Yaskawa INFORM job: test_long_tjr6.JBI

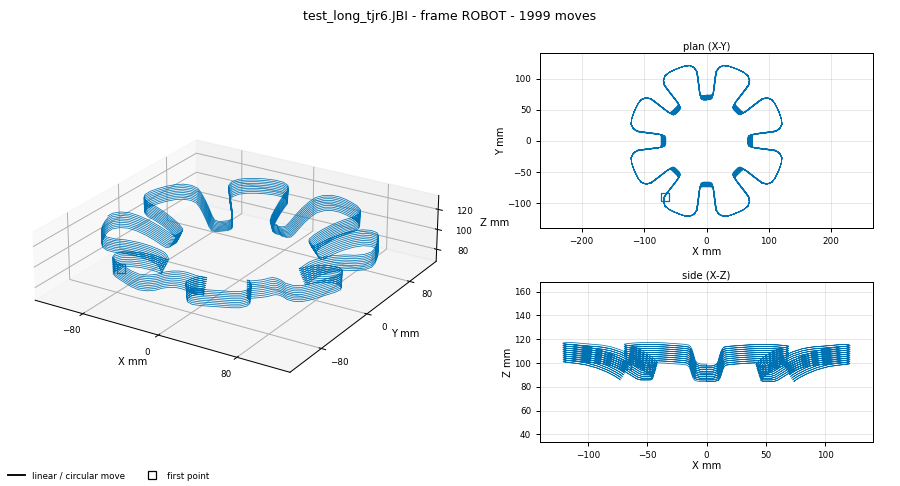
[picture p0: tool path of test_long_tjr6.JBI in frame ROBOT, 1999 of 2000 moves have a stored position in this frame; points joined in program order, loops and branches not executed]
version: 0
/JOB
//NAME test_long
//POS
///NPOS 48,0,0,2,0,0
///TOOL 1
///POSTYPE ROBOT
///RECTAN
///RCONF 1,0,0,0,0,0,0,0,0,0,0,0,0,0,0,0,0,0,0,0,0,0,0,0
C00000=-62.110,-83.210,96.990,-0.0900,0.0600,0.9900
C00001=-67.170,-90.300,98.220,-0.0900,0.0500,0.9900
C00002=-68.520,-97.840,98.870,-0.0700,-0.0100,1.0000
C00003=-65.820,-104.830,99.390,-0.0300,-0.0200,1.0000
C00004=-59.610,-109.840,99.910,-0.0000,-0.0000,1.0000
C00005=-51.890,-113.720,100.250,-0.0000,-0.0000,1.0000
C00006=-43.720,-117.100,100.250,-0.0000,-0.0000,1.0000
C00007=-35.520,-119.820,99.910,-0.0000,-0.0000,1.0000
C00008=-27.590,-120.670,99.390,0.0000,-0.0300,1.0000
C00009=-20.730,-117.630,98.870,0.0400,-0.0500,1.0000
C00010=-16.350,-111.350,98.220,0.1000,-0.0300,0.9900
C00011=-14.920,-102.760,96.990,0.1000,-0.0200,0.9900
C00012=-13.710,-93.380,94.450,0.0900,-0.0100,1.0000
C00013=-12.630,-84.870,91.070,0.0700,-0.0100,1.0000
C00014=-11.600,-78.400,87.740,0.0300,-0.0100,1.0000
C00015=-9.810,-74.590,85.320,-0.2400,0.2600,0.9300
C00016=-5.850,-73.580,84.360,-0.0500,0.5500,0.8400
C00017=-2.550,-73.670,84.320,0.0200,0.5600,0.8300
C00018=0.000,-73.710,84.350,-0.0000,0.5600,0.8300
C00019=0.000,-73.710,84.350,-0.0000,0.5600,0.8300
C00020=2.550,-73.670,84.320,-0.0200,0.5600,0.8300
C00021=5.850,-73.580,84.360,0.0500,0.5500,0.8400
C00022=9.810,-74.580,85.320,0.2400,0.2600,0.9300
C00023=11.600,-78.400,87.740,-0.0300,-0.0100,1.0000
C00024=12.630,-84.870,91.070,-0.0700,-0.0100,1.0000
C00025=13.710,-93.380,94.450,-0.0900,-0.0100,1.0000
C00026=14.920,-102.760,96.990,-0.1000,-0.0200,0.9900
C00027=16.350,-111.350,98.220,-0.1000,-0.0300,0.9900
C00028=20.730,-117.630,98.870,-0.0400,-0.0500,1.0000
C00029=27.590,-120.670,99.390,-0.0000,-0.0300,1.0000
C00030=35.520,-119.820,99.910,0.0000,-0.0000,1.0000
C00031=43.720,-117.100,100.250,0.0000,-0.0000,1.0000
C00032=51.890,-113.720,100.250,0.0000,-0.0000,1.0000
C00033=59.610,-109.840,99.910,0.0000,-0.0000,1.0000
C00034=65.820,-104.830,99.390,0.0300,-0.0200,1.0000
C00035=68.520,-97.840,98.870,0.0700,-0.0100,1.0000
C00036=67.170,-90.300,98.220,0.0900,0.0500,0.9900
C00037=62.110,-83.210,96.990,0.0900,0.0600,0.9900
C00038=56.330,-75.720,94.450,0.0800,0.0600,1.0000
C00039=51.080,-68.940,91.070,0.0600,0.0400,1.0000
C00040=47.240,-63.640,87.740,0.0200,0.0100,1.0000
C00041=45.800,-59.680,85.320,-0.3600,0.0200,0.9300
C00042=47.890,-56.170,84.360,-0.4200,0.3500,0.8400
C00043=50.290,-53.900,84.320,-0.3800,0.4100,0.8300
C00044=52.120,-52.120,84.350,-0.4000,0.4000,0.8300
C00045=53.900,-50.290,84.320,-0.4100,0.3800,0.8300
C00046=56.170,-47.890,84.360,-0.3500,0.4200,0.8400
C00047=59.680,-45.800,85.320,-0.0200,0.3600,0.9300
C00048=63.640,-47.240,87.740,-0.0100,-0.0200,1.0000
C00049=68.940,-51.080,91.070,-0.0400,-0.0600,1.0000
C00050=75.720,-56.330,94.450,-0.0600,-0.0800,1.0000
C00051=83.210,-62.110,96.990,-0.0600,-0.0900,0.9900
C00052=90.300,-67.170,98.220,-0.0500,-0.0900,0.9900
C00053=97.840,-68.520,98.870,0.0100,-0.0700,1.0000
C00054=104.830,-65.820,99.390,0.0200,-0.0300,1.0000
C00055=109.840,-59.610,99.910,0.0000,-0.0000,1.0000
C00056=113.720,-51.890,100.250,0.0000,-0.0000,1.0000
C00057=117.100,-43.720,100.250,0.0000,-0.0000,1.0000
C00058=119.820,-35.520,99.910,0.0000,-0.0000,1.0000
C00059=120.670,-27.590,99.390,0.0300,0.0000,1.0000
C00060=117.630,-20.730,98.870,0.0500,0.0400,1.0000
C00061=111.350,-16.350,98.220,0.0300,0.1000,0.9900
C00062=102.760,-14.920,96.990,0.0200,0.1000,0.9900
C00063=93.380,-13.710,94.450,0.0100,0.0900,1.0000
C00064=84.870,-12.630,91.070,0.0100,0.0700,1.0000
C00065=78.400,-11.600,87.740,0.0100,0.0300,1.0000
C00066=74.590,-9.810,85.320,-0.2600,-0.2400,0.9300
C00067=73.580,-5.850,84.360,-0.5500,-0.0500,0.8400
C00068=73.670,-2.550,84.320,-0.5600,0.0200,0.8300
C00069=73.710,0.000,84.350,-0.5600,-0.0000,0.8300
C00070=73.670,2.550,84.320,-0.5600,-0.0200,0.8300
C00071=73.580,5.850,84.360,-0.5500,0.0500,0.8400
C00072=74.580,9.810,85.320,-0.2600,0.2400,0.9300
C00073=78.400,11.600,87.740,0.0100,-0.0300,1.0000
C00074=84.870,12.630,91.070,0.0100,-0.0700,1.0000
C00075=93.380,13.710,94.450,0.0100,-0.0900,1.0000
C00076=102.760,14.920,96.990,0.0200,-0.1000,0.9900
C00077=111.350,16.350,98.220,0.0300,-0.1000,0.9900
C00078=117.630,20.730,98.870,0.0500,-0.0400,1.0000
C00079=120.670,27.590,99.390,0.0300,-0.0000,1.0000
C00080=119.820,35.520,99.910,0.0000,0.0000,1.0000
C00081=117.100,43.720,100.250,0.0000,0.0000,1.0000
C00082=113.720,51.890,100.250,0.0000,0.0000,1.0000
C00083=109.840,59.610,99.910,0.0000,0.0000,1.0000
C00084=104.830,65.820,99.390,0.0200,0.0300,1.0000
C00085=97.840,68.520,98.870,0.0100,0.0700,1.0000
C00086=90.300,67.170,98.220,-0.0500,0.0900,0.9900
C00087=83.210,62.110,96.990,-0.0600,0.0900,0.9900
C00088=75.720,56.330,94.450,-0.0600,0.0800,1.0000
C00089=68.940,51.080,91.070,-0.0400,0.0600,1.0000
C00090=63.640,47.240,87.740,-0.0100,0.0200,1.0000
C00091=59.680,45.800,85.320,-0.0200,-0.3600,0.9300
C00092=56.170,47.890,84.360,-0.3500,-0.4200,0.8400
C00093=53.900,50.290,84.320,-0.4100,-0.3800,0.8300
C00094=52.120,52.120,84.350,-0.4000,-0.4000,0.8300
C00095=50.290,53.900,84.320,-0.3800,-0.4100,0.8300
C00096=47.890,56.170,84.360,-0.4200,-0.3500,0.8400
C00097=45.800,59.680,85.320,-0.3600,-0.0200,0.9300
C00098=47.240,63.640,87.740,0.0200,-0.0100,1.0000
C00099=51.080,68.940,91.070,0.0600,-0.0400,1.0000
C00100=56.330,75.720,94.450,0.0800,-0.0600,1.0000
C00101=62.110,83.210,96.990,0.0900,-0.0600,0.9900
C00102=67.170,90.300,98.220,0.0900,-0.0500,0.9900
C00103=68.520,97.840,98.870,0.0700,0.0100,1.0000
C00104=65.820,104.830,99.390,0.0300,0.0200,1.0000
C00105=59.610,109.840,99.910,0.0000,0.0000,1.0000
C00106=51.890,113.720,100.250,0.0000,0.0000,1.0000
C00107=43.720,117.100,100.250,0.0000,0.0000,1.0000
C00108=35.520,119.820,99.910,0.0000,0.0000,1.0000
C00109=27.590,120.670,99.390,-0.0000,0.0300,1.0000
C00110=20.730,117.630,98.870,-0.0400,0.0500,1.0000
C00111=16.350,111.350,98.220,-0.1000,0.0300,0.9900
C00112=14.920,102.760,96.990,-0.1000,0.0200,0.9900
C00113=13.710,93.380,94.450,-0.0900,0.0100,1.0000
C00114=12.630,84.870,91.070,-0.0700,0.0100,1.0000
C00115=11.600,78.400,87.740,-0.0300,0.0100,1.0000
C00116=9.810,74.580,85.320,0.2400,-0.2600,0.9300
C00117=5.850,73.580,84.360,0.0500,-0.5500,0.8400
C00118=2.550,73.670,84.320,-0.0200,-0.5600,0.8300
C00119=0.000,73.710,84.350,-0.0000,-0.5600,0.8300
C00120=0.000,72.760,85.760,-0.0000,-0.5500,0.8300
C00121=2.470,72.730,85.730,-0.0200,-0.5500,0.8300
C00122=5.710,72.650,85.770,0.0500,-0.5400,0.8400
C00123=9.640,73.690,86.760,0.2300,-0.2500,0.9400
C00124=11.390,77.620,89.240,-0.0300,0.0100,1.0000
C00125=12.400,84.250,92.640,-0.0700,0.0100,1.0000
C00126=13.490,92.950,96.080,-0.0900,0.0100,1.0000
C00127=14.700,102.500,98.660,-0.1000,0.0200,0.9900
C00128=16.130,111.230,99.900,-0.0900,0.0300,1.0000
C00129=20.530,117.600,100.550,-0.0400,0.0500,1.0000
C00130=27.430,120.700,101.080,-0.0000,0.0300,1.0000
C00131=35.420,119.860,101.610,0.0000,0.0000,1.0000
C00132=43.690,117.110,101.950,0.0000,0.0000,1.0000
C00133=51.920,113.700,101.950,0.0000,0.0000,1.0000
C00134=59.710,109.800,101.610,0.0000,0.0000,1.0000
C00135=65.950,104.740,101.080,0.0200,0.0200,1.0000
C00136=68.640,97.670,100.550,0.0600,0.0100,1.0000
C00137=67.240,90.060,99.900,0.0900,-0.0400,1.0000
C00138=62.080,82.880,98.660,0.0800,-0.0600,0.9900
C00139=56.180,75.270,96.080,0.0700,-0.0500,1.0000
C00140=50.810,68.350,92.640,0.0600,-0.0400,1.0000
C00141=46.830,62.940,89.240,0.0200,-0.0200,1.0000
C00142=45.290,58.920,86.760,-0.3400,-0.0100,0.9400
C00143=47.330,55.400,85.770,-0.4200,-0.3400,0.8400
C00144=49.680,53.170,85.730,-0.3700,-0.4100,0.8300
C00145=51.450,51.450,85.760,-0.3900,-0.3900,0.8300
C00146=53.170,49.680,85.730,-0.4100,-0.3700,0.8300
C00147=55.400,47.330,85.770,-0.3400,-0.4200,0.8400
C00148=58.920,45.290,86.760,-0.0100,-0.3400,0.9400
C00149=62.940,46.830,89.240,-0.0200,0.0200,1.0000
C00150=68.350,50.810,92.640,-0.0400,0.0600,1.0000
C00151=75.270,56.180,96.080,-0.0500,0.0700,1.0000
C00152=82.880,62.080,98.660,-0.0600,0.0800,0.9900
C00153=90.060,67.240,99.900,-0.0400,0.0900,1.0000
C00154=97.670,68.640,100.550,0.0100,0.0600,1.0000
C00155=104.740,65.950,101.080,0.0200,0.0200,1.0000
C00156=109.800,59.710,101.610,0.0000,0.0000,1.0000
C00157=113.700,51.920,101.950,0.0000,0.0000,1.0000
C00158=117.110,43.690,101.950,0.0000,0.0000,1.0000
C00159=119.860,35.420,101.610,0.0000,0.0000,1.0000
C00160=120.700,27.430,101.080,0.0300,-0.0000,1.0000
C00161=117.600,20.530,100.550,0.0500,-0.0400,1.0000
C00162=111.230,16.130,99.900,0.0300,-0.0900,1.0000
C00163=102.500,14.700,98.660,0.0200,-0.1000,0.9900
C00164=92.950,13.490,96.080,0.0100,-0.0900,1.0000
C00165=84.250,12.400,92.640,0.0100,-0.0700,1.0000
C00166=77.620,11.390,89.240,0.0100,-0.0300,1.0000
C00167=73.690,9.640,86.760,-0.2500,0.2300,0.9400
C00168=72.650,5.710,85.770,-0.5400,0.0500,0.8400
C00169=72.730,2.470,85.730,-0.5500,-0.0200,0.8300
C00170=72.760,0.000,85.760,-0.5500,-0.0000,0.8300
C00171=72.730,-2.470,85.730,-0.5500,0.0200,0.8300
C00172=72.650,-5.710,85.770,-0.5400,-0.0500,0.8400
C00173=73.690,-9.640,86.760,-0.2500,-0.2300,0.9400
C00174=77.620,-11.390,89.240,0.0100,0.0300,1.0000
C00175=84.250,-12.400,92.640,0.0100,0.0700,1.0000
C00176=92.950,-13.490,96.080,0.0100,0.0900,1.0000
C00177=102.500,-14.700,98.660,0.0200,0.1000,0.9900
C00178=111.230,-16.130,99.900,0.0300,0.0900,1.0000
C00179=117.600,-20.530,100.550,0.0500,0.0400,1.0000
C00180=120.700,-27.430,101.080,0.0300,0.0000,1.0000
C00181=119.860,-35.420,101.610,0.0000,-0.0000,1.0000
C00182=117.110,-43.690,101.950,0.0000,-0.0000,1.0000
C00183=113.700,-51.920,101.950,0.0000,-0.0000,1.0000
C00184=109.800,-59.710,101.610,0.0000,-0.0000,1.0000
C00185=104.740,-65.950,101.080,0.0200,-0.0200,1.0000
C00186=97.670,-68.640,100.550,0.0100,-0.0600,1.0000
C00187=90.060,-67.240,99.900,-0.0400,-0.0900,1.0000
C00188=82.880,-62.080,98.660,-0.0600,-0.0800,0.9900
C00189=75.270,-56.180,96.080,-0.0500,-0.0700,1.0000
C00190=68.350,-50.810,92.640,-0.0400,-0.0600,1.0000
C00191=62.940,-46.830,89.240,-0.0200,-0.0200,1.0000
C00192=58.920,-45.290,86.760,-0.0100,0.3400,0.9400
C00193=55.400,-47.330,85.770,-0.3400,0.4200,0.8400
C00194=53.170,-49.680,85.730,-0.4100,0.3700,0.8300
C00195=51.450,-51.450,85.760,-0.3900,0.3900,0.8300
C00196=49.680,-53.170,85.730,-0.3700,0.4100,0.8300
C00197=47.330,-55.400,85.770,-0.4200,0.3400,0.8400
C00198=45.290,-58.920,86.760,-0.3400,0.0100,0.9400
C00199=46.830,-62.940,89.240,0.0200,0.0200,1.0000
C00200=50.810,-68.350,92.640,0.0600,0.0400,1.0000
C00201=56.180,-75.270,96.080,0.0700,0.0500,1.0000
C00202=62.080,-82.880,98.660,0.0800,0.0600,0.9900
C00203=67.240,-90.060,99.900,0.0900,0.0400,1.0000
C00204=68.640,-97.670,100.550,0.0600,-0.0100,1.0000
C00205=65.950,-104.740,101.080,0.0200,-0.0200,1.0000
C00206=59.710,-109.800,101.610,0.0000,-0.0000,1.0000
C00207=51.920,-113.700,101.950,0.0000,-0.0000,1.0000
C00208=43.690,-117.110,101.950,0.0000,-0.0000,1.0000
C00209=35.420,-119.860,101.610,0.0000,-0.0000,1.0000
C00210=27.430,-120.700,101.080,-0.0000,-0.0300,1.0000
C00211=20.530,-117.600,100.550,-0.0400,-0.0500,1.0000
C00212=16.130,-111.230,99.900,-0.0900,-0.0300,1.0000
C00213=14.700,-102.500,98.660,-0.1000,-0.0200,0.9900
C00214=13.490,-92.950,96.080,-0.0900,-0.0100,1.0000
C00215=12.400,-84.250,92.640,-0.0700,-0.0100,1.0000
C00216=11.390,-77.620,89.240,-0.0300,-0.0100,1.0000
C00217=9.640,-73.690,86.760,0.2300,0.2500,0.9400
C00218=5.710,-72.650,85.770,0.0500,0.5400,0.8400
C00219=2.470,-72.730,85.730,-0.0200,0.5500,0.8300
C00220=0.000,-72.760,85.760,-0.0000,0.5500,0.8300
C00221=0.000,-72.760,85.760,-0.0000,0.5500,0.8300
C00222=-2.470,-72.730,85.730,0.0200,0.5500,0.8300
C00223=-5.710,-72.650,85.770,-0.0500,0.5400,0.8400
C00224=-9.640,-73.690,86.760,-0.2300,0.2500,0.9400
C00225=-11.390,-77.620,89.240,0.0300,-0.0100,1.0000
C00226=-12.400,-84.250,92.640,0.0700,-0.0100,1.0000
C00227=-13.490,-92.950,96.080,0.0900,-0.0100,1.0000
C00228=-14.700,-102.500,98.660,0.1000,-0.0200,0.9900
C00229=-16.130,-111.230,99.900,0.0900,-0.0300,1.0000
C00230=-20.530,-117.600,100.550,0.0400,-0.0500,1.0000
C00231=-27.430,-120.700,101.080,0.0000,-0.0300,1.0000
C00232=-35.420,-119.860,101.610,-0.0000,-0.0000,1.0000
C00233=-43.690,-117.110,101.950,-0.0000,-0.0000,1.0000
C00234=-51.920,-113.700,101.950,-0.0000,-0.0000,1.0000
C00235=-59.710,-109.800,101.610,-0.0000,-0.0000,1.0000
C00236=-65.950,-104.740,101.080,-0.0200,-0.0200,1.0000
C00237=-68.640,-97.670,100.550,-0.0600,-0.0100,1.0000
C00238=-67.240,-90.060,99.900,-0.0900,0.0400,1.0000
C00239=-62.080,-82.880,98.660,-0.0800,0.0600,0.9900
C00240=-56.180,-75.270,96.080,-0.0700,0.0500,1.0000
C00241=-50.810,-68.350,92.640,-0.0600,0.0400,1.0000
C00242=-46.830,-62.940,89.240,-0.0200,0.0200,1.0000
C00243=-45.290,-58.920,86.760,0.3400,0.0100,0.9400
C00244=-47.330,-55.400,85.770,0.4200,0.3400,0.8400
C00245=-49.680,-53.170,85.730,0.3700,0.4100,0.8300
C00246=-51.450,-51.450,85.760,0.3900,0.3900,0.8300
C00247=-53.170,-49.680,85.730,0.4100,0.3700,0.8300
C00248=-55.400,-47.330,85.770,0.3400,0.4200,0.8400
C00249=-58.920,-45.290,86.760,0.0100,0.3400,0.9400
C00250=-62.940,-46.830,89.240,0.0200,-0.0200,1.0000
C00251=-68.350,-50.810,92.640,0.0400,-0.0600,1.0000
C00252=-75.270,-56.180,96.080,0.0500,-0.0700,1.0000
C00253=-82.880,-62.080,98.660,0.0600,-0.0800,0.9900
C00254=-90.060,-67.240,99.900,0.0400,-0.0900,1.0000
C00255=-97.670,-68.640,100.550,-0.0100,-0.0600,1.0000
C00256=-104.740,-65.950,101.080,-0.0200,-0.0200,1.0000
C00257=-109.800,-59.710,101.610,-0.0000,-0.0000,1.0000
C00258=-113.700,-51.920,101.950,-0.0000,-0.0000,1.0000
C00259=-117.110,-43.690,101.950,-0.0000,-0.0000,1.0000
C00260=-119.860,-35.420,101.610,-0.0000,-0.0000,1.0000
C00261=-120.700,-27.430,101.080,-0.0300,0.0000,1.0000
C00262=-117.600,-20.530,100.550,-0.0500,0.0400,1.0000
C00263=-111.230,-16.130,99.900,-0.0300,0.0900,1.0000
C00264=-102.500,-14.700,98.660,-0.0200,0.1000,0.9900
C00265=-92.950,-13.490,96.080,-0.0100,0.0900,1.0000
C00266=-84.250,-12.400,92.640,-0.0100,0.0700,1.0000
C00267=-77.620,-11.390,89.240,-0.0100,0.0300,1.0000
C00268=-73.690,-9.640,86.760,0.2500,-0.2300,0.9400
C00269=-72.650,-5.710,85.770,0.5400,-0.0500,0.8400
C00270=-72.730,-2.470,85.730,0.5500,0.0200,0.8300
C00271=-72.760,0.000,85.760,0.5500,0.0000,0.8300
C00272=-72.730,2.470,85.730,0.5500,-0.0200,0.8300
C00273=-72.650,5.710,85.770,0.5400,0.0500,0.8400
C00274=-73.690,9.640,86.760,0.2500,0.2300,0.9400
C00275=-77.620,11.390,89.240,-0.0100,-0.0300,1.0000
C00276=-84.250,12.400,92.640,-0.0100,-0.0700,1.0000
C00277=-92.950,13.490,96.080,-0.0100,-0.0900,1.0000
C00278=-102.500,14.700,98.660,-0.0200,-0.1000,0.9900
C00279=-111.230,16.130,99.900,-0.0300,-0.0900,1.0000
C00280=-117.600,20.530,100.550,-0.0500,-0.0400,1.0000
C00281=-120.700,27.430,101.080,-0.0300,-0.0000,1.0000
C00282=-119.860,35.420,101.610,-0.0000,0.0000,1.0000
C00283=-117.110,43.690,101.950,-0.0000,0.0000,1.0000
C00284=-113.700,51.920,101.950,-0.0000,0.0000,1.0000
C00285=-109.800,59.710,101.610,-0.0000,0.0000,1.0000
C00286=-104.740,65.950,101.080,-0.0200,0.0200,1.0000
C00287=-97.670,68.640,100.550,-0.0100,0.0600,1.0000
C00288=-90.060,67.240,99.900,0.0400,0.0900,1.0000
C00289=-82.880,62.080,98.660,0.0600,0.0800,0.9900
C00290=-75.270,56.180,96.080,0.0500,0.0700,1.0000
C00291=-68.350,50.810,92.640,0.0400,0.0600,1.0000
C00292=-62.940,46.830,89.240,0.0200,0.0200,1.0000
C00293=-58.920,45.290,86.760,0.0100,-0.3400,0.9400
C00294=-55.400,47.330,85.770,0.3400,-0.4200,0.8400
C00295=-53.170,49.680,85.730,0.4100,-0.3700,0.8300
C00296=-51.450,51.450,85.760,0.3900,-0.3900,0.8300
C00297=-49.680,53.170,85.730,0.3700,-0.4100,0.8300
C00298=-47.330,55.400,85.770,0.4200,-0.3400,0.8400
C00299=-45.290,58.920,86.760,0.3400,-0.0100,0.9400
C00300=-46.830,62.940,89.240,-0.0200,-0.0200,1.0000
C00301=-50.810,68.350,92.640,-0.0600,-0.0400,1.0000
C00302=-56.180,75.270,96.080,-0.0700,-0.0500,1.0000
C00303=-62.080,82.880,98.660,-0.0800,-0.0600,0.9900
C00304=-67.240,90.060,99.900,-0.0900,-0.0400,1.0000
C00305=-68.640,97.670,100.550,-0.0600,0.0100,1.0000
C00306=-65.950,104.740,101.080,-0.0200,0.0200,1.0000
C00307=-59.710,109.800,101.610,-0.0000,0.0000,1.0000
C00308=-51.920,113.700,101.950,-0.0000,0.0000,1.0000
C00309=-43.690,117.110,101.950,-0.0000,0.0000,1.0000
C00310=-35.420,119.860,101.610,-0.0000,0.0000,1.0000
C00311=-27.430,120.700,101.080,0.0000,0.0300,1.0000
C00312=-20.530,117.600,100.550,0.0400,0.0500,1.0000
C00313=-16.130,111.230,99.900,0.0900,0.0300,1.0000
C00314=-14.700,102.500,98.660,0.1000,0.0200,0.9900
C00315=-13.490,92.950,96.080,0.0900,0.0100,1.0000
C00316=-12.400,84.250,92.640,0.0700,0.0100,1.0000
C00317=-11.390,77.620,89.240,0.0300,0.0100,1.0000
C00318=-9.640,73.690,86.760,-0.2300,-0.2500,0.9400
C00319=-5.710,72.650,85.770,-0.0500,-0.5400,0.8400
C00320=-2.470,72.730,85.730,0.0200,-0.5500,0.8300
C00321=0.000,72.760,85.760,-0.0000,-0.5500,0.8300
C00322=0.000,71.830,87.180,-0.0000,-0.5400,0.8400
C00323=-2.380,71.800,87.150,0.0200,-0.5400,0.8400
C00324=-5.560,71.730,87.200,-0.0500,-0.5300,0.8500
C00325=-9.460,72.820,88.210,-0.2300,-0.2400,0.9400
C00326=-11.190,76.860,90.740,0.0300,0.0100,1.0000
C00327=-12.190,83.660,94.220,0.0700,0.0100,1.0000
C00328=-13.290,92.540,97.720,0.0900,0.0100,1.0000
C00329=-14.500,102.260,100.330,0.0900,0.0100,1.0000
C00330=-15.920,111.110,101.590,0.0900,0.0300,1.0000
C00331=-20.340,117.580,102.240,0.0400,0.0500,1.0000
C00332=-27.280,120.720,102.770,0.0000,0.0300,1.0000
C00333=-35.330,119.890,103.300,-0.0000,0.0000,1.0000
C00334=-43.660,117.130,103.650,-0.0000,0.0000,1.0000
C00335=-51.950,113.690,103.650,-0.0000,0.0000,1.0000
C00336=-59.790,109.750,103.300,-0.0000,0.0000,1.0000
C00337=-66.070,104.660,102.770,-0.0200,0.0200,1.0000
C00338=-68.760,97.520,102.240,-0.0600,0.0100,1.0000
C00339=-67.310,89.830,101.590,-0.0800,-0.0400,1.0000
C00340=-62.060,82.560,100.330,-0.0800,-0.0600,1.0000
C00341=-56.040,74.830,97.720,-0.0700,-0.0500,1.0000
C00342=-50.540,67.780,94.220,-0.0600,-0.0400,1.0000
C00343=-46.440,62.260,90.740,-0.0300,-0.0200,1.0000
C00344=-44.800,58.180,88.210,0.3300,-0.0100,0.9400
C00345=-46.780,54.650,87.200,0.4100,-0.3300,0.8500
C00346=-49.090,52.450,87.150,0.3700,-0.4000,0.8400
C00347=-50.790,50.790,87.180,0.3800,-0.3800,0.8400
C00348=-52.450,49.090,87.150,0.4000,-0.3700,0.8400
C00349=-54.650,46.780,87.200,0.3300,-0.4100,0.8500
C00350=-58.180,44.800,88.210,0.0100,-0.3300,0.9400
C00351=-62.260,46.440,90.740,0.0200,0.0300,1.0000
C00352=-67.780,50.540,94.220,0.0400,0.0600,1.0000
C00353=-74.830,56.040,97.720,0.0500,0.0700,1.0000
C00354=-82.560,62.060,100.330,0.0600,0.0800,1.0000
C00355=-89.830,67.310,101.590,0.0400,0.0800,1.0000
C00356=-97.520,68.760,102.240,-0.0100,0.0600,1.0000
C00357=-104.660,66.070,102.770,-0.0200,0.0200,1.0000
C00358=-109.750,59.790,103.300,-0.0000,0.0000,1.0000
C00359=-113.690,51.950,103.650,-0.0000,0.0000,1.0000
C00360=-117.130,43.660,103.650,-0.0000,0.0000,1.0000
C00361=-119.890,35.330,103.300,-0.0000,0.0000,1.0000
C00362=-120.720,27.280,102.770,-0.0300,-0.0000,1.0000
C00363=-117.580,20.340,102.240,-0.0500,-0.0400,1.0000
C00364=-111.110,15.920,101.590,-0.0300,-0.0900,1.0000
C00365=-102.260,14.500,100.330,-0.0100,-0.0900,1.0000
C00366=-92.540,13.290,97.720,-0.0100,-0.0900,1.0000
C00367=-83.660,12.190,94.220,-0.0100,-0.0700,1.0000
C00368=-76.860,11.190,90.740,-0.0100,-0.0300,1.0000
C00369=-72.820,9.460,88.210,0.2400,0.2300,0.9400
C00370=-71.730,5.560,87.200,0.5300,0.0500,0.8500
C00371=-71.800,2.380,87.150,0.5400,-0.0200,0.8400
C00372=-71.830,0.000,87.180,0.5400,0.0000,0.8400
C00373=-71.800,-2.380,87.150,0.5400,0.0200,0.8400
C00374=-71.730,-5.560,87.200,0.5300,-0.0500,0.8500
C00375=-72.820,-9.460,88.210,0.2400,-0.2300,0.9400
C00376=-76.860,-11.190,90.740,-0.0100,0.0300,1.0000
C00377=-83.660,-12.190,94.220,-0.0100,0.0700,1.0000
C00378=-92.540,-13.290,97.720,-0.0100,0.0900,1.0000
C00379=-102.260,-14.500,100.330,-0.0100,0.0900,1.0000
C00380=-111.110,-15.920,101.590,-0.0300,0.0900,1.0000
C00381=-117.580,-20.340,102.240,-0.0500,0.0400,1.0000
C00382=-120.720,-27.280,102.770,-0.0300,0.0000,1.0000
C00383=-119.890,-35.330,103.300,-0.0000,-0.0000,1.0000
C00384=-117.130,-43.660,103.650,-0.0000,-0.0000,1.0000
C00385=-113.690,-51.950,103.650,-0.0000,-0.0000,1.0000
C00386=-109.750,-59.790,103.300,-0.0000,-0.0000,1.0000
C00387=-104.660,-66.070,102.770,-0.0200,-0.0200,1.0000
C00388=-97.520,-68.760,102.240,-0.0100,-0.0600,1.0000
C00389=-89.830,-67.310,101.590,0.0400,-0.0800,1.0000
C00390=-82.560,-62.060,100.330,0.0600,-0.0800,1.0000
C00391=-74.830,-56.040,97.720,0.0500,-0.0700,1.0000
C00392=-67.780,-50.540,94.220,0.0400,-0.0600,1.0000
C00393=-62.260,-46.440,90.740,0.0200,-0.0300,1.0000
C00394=-58.180,-44.800,88.210,0.0100,0.3300,0.9400
C00395=-54.650,-46.780,87.200,0.3300,0.4100,0.8500
C00396=-52.450,-49.090,87.150,0.4000,0.3700,0.8400
C00397=-50.790,-50.790,87.180,0.3800,0.3800,0.8400
C00398=-49.090,-52.450,87.150,0.3700,0.4000,0.8400
C00399=-46.780,-54.650,87.200,0.4100,0.3300,0.8500
C00400=-44.800,-58.180,88.210,0.3300,0.0100,0.9400
C00401=-46.440,-62.260,90.740,-0.0300,0.0200,1.0000
C00402=-50.540,-67.780,94.220,-0.0600,0.0400,1.0000
C00403=-56.040,-74.830,97.720,-0.0700,0.0500,1.0000
C00404=-62.060,-82.560,100.330,-0.0800,0.0600,1.0000
C00405=-67.310,-89.830,101.590,-0.0800,0.0400,1.0000
C00406=-68.760,-97.520,102.240,-0.0600,-0.0100,1.0000
C00407=-66.070,-104.660,102.770,-0.0200,-0.0200,1.0000
C00408=-59.790,-109.750,103.300,-0.0000,-0.0000,1.0000
C00409=-51.950,-113.690,103.650,-0.0000,-0.0000,1.0000
C00410=-43.660,-117.130,103.650,-0.0000,-0.0000,1.0000
C00411=-35.330,-119.890,103.300,-0.0000,-0.0000,1.0000
C00412=-27.280,-120.720,102.770,0.0000,-0.0300,1.0000
C00413=-20.340,-117.580,102.240,0.0400,-0.0500,1.0000
C00414=-15.920,-111.110,101.590,0.0900,-0.0300,1.0000
C00415=-14.500,-102.260,100.330,0.0900,-0.0100,1.0000
C00416=-13.290,-92.540,97.720,0.0900,-0.0100,1.0000
C00417=-12.190,-83.660,94.220,0.0700,-0.0100,1.0000
C00418=-11.190,-76.860,90.740,0.0300,-0.0100,1.0000
C00419=-9.460,-72.820,88.210,-0.2300,0.2400,0.9400
C00420=-5.560,-71.730,87.200,-0.0500,0.5300,0.8500
C00421=-2.380,-71.800,87.150,0.0200,0.5400,0.8400
C00422=0.000,-71.830,87.180,-0.0000,0.5400,0.8400
C00423=0.000,-71.830,87.180,-0.0000,0.5400,0.8400
C00424=2.380,-71.800,87.150,-0.0200,0.5400,0.8400
C00425=5.560,-71.730,87.200,0.0500,0.5300,0.8500
C00426=9.460,-72.820,88.210,0.2300,0.2400,0.9400
C00427=11.190,-76.860,90.740,-0.0300,-0.0100,1.0000
C00428=12.190,-83.660,94.220,-0.0700,-0.0100,1.0000
C00429=13.290,-92.540,97.720,-0.0900,-0.0100,1.0000
C00430=14.500,-102.260,100.330,-0.0900,-0.0100,1.0000
C00431=15.920,-111.110,101.590,-0.0900,-0.0300,1.0000
C00432=20.340,-117.580,102.240,-0.0400,-0.0500,1.0000
C00433=27.280,-120.720,102.770,-0.0000,-0.0300,1.0000
C00434=35.330,-119.890,103.300,0.0000,-0.0000,1.0000
C00435=43.660,-117.130,103.650,0.0000,-0.0000,1.0000
C00436=51.950,-113.690,103.650,0.0000,-0.0000,1.0000
C00437=59.790,-109.750,103.300,0.0000,-0.0000,1.0000
C00438=66.070,-104.660,102.770,0.0200,-0.0200,1.0000
C00439=68.760,-97.520,102.240,0.0600,-0.0100,1.0000
C00440=67.310,-89.830,101.590,0.0800,0.0400,1.0000
C00441=62.060,-82.560,100.330,0.0800,0.0600,1.0000
C00442=56.040,-74.830,97.720,0.0700,0.0500,1.0000
C00443=50.540,-67.780,94.220,0.0600,0.0400,1.0000
C00444=46.440,-62.260,90.740,0.0300,0.0200,1.0000
C00445=44.800,-58.180,88.210,-0.3300,0.0100,0.9400
C00446=46.780,-54.650,87.200,-0.4100,0.3300,0.8500
C00447=49.090,-52.450,87.150,-0.3700,0.4000,0.8400
C00448=50.790,-50.790,87.180,-0.3800,0.3800,0.8400
C00449=52.450,-49.090,87.150,-0.4000,0.3700,0.8400
C00450=54.650,-46.780,87.200,-0.3300,0.4100,0.8500
C00451=58.180,-44.800,88.210,-0.0100,0.3300,0.9400
C00452=62.260,-46.440,90.740,-0.0200,-0.0300,1.0000
C00453=67.780,-50.540,94.220,-0.0400,-0.0600,1.0000
C00454=74.830,-56.040,97.720,-0.0500,-0.0700,1.0000
C00455=82.560,-62.060,100.330,-0.0600,-0.0800,1.0000
C00456=89.830,-67.310,101.590,-0.0400,-0.0800,1.0000
C00457=97.520,-68.760,102.240,0.0100,-0.0600,1.0000
C00458=104.660,-66.070,102.770,0.0200,-0.0200,1.0000
C00459=109.750,-59.790,103.300,0.0000,-0.0000,1.0000
C00460=113.690,-51.950,103.650,0.0000,-0.0000,1.0000
C00461=117.130,-43.660,103.650,0.0000,-0.0000,1.0000
C00462=119.890,-35.330,103.300,0.0000,-0.0000,1.0000
C00463=120.720,-27.280,102.770,0.0300,0.0000,1.0000
C00464=117.580,-20.340,102.240,0.0500,0.0400,1.0000
C00465=111.110,-15.920,101.590,0.0300,0.0900,1.0000
C00466=102.260,-14.500,100.330,0.0100,0.0900,1.0000
C00467=92.540,-13.290,97.720,0.0100,0.0900,1.0000
C00468=83.660,-12.190,94.220,0.0100,0.0700,1.0000
C00469=76.860,-11.190,90.740,0.0100,0.0300,1.0000
C00470=72.820,-9.460,88.210,-0.2400,-0.2300,0.9400
C00471=71.730,-5.560,87.200,-0.5300,-0.0500,0.8500
C00472=71.800,-2.380,87.150,-0.5400,0.0200,0.8400
C00473=71.830,0.000,87.180,-0.5400,-0.0000,0.8400
C00474=71.800,2.380,87.150,-0.5400,-0.0200,0.8400
C00475=71.730,5.560,87.200,-0.5300,0.0500,0.8500
C00476=72.820,9.460,88.210,-0.2400,0.2300,0.9400
C00477=76.860,11.190,90.740,0.0100,-0.0300,1.0000
C00478=83.660,12.190,94.220,0.0100,-0.0700,1.0000
C00479=92.540,13.290,97.720,0.0100,-0.0900,1.0000
C00480=102.260,14.500,100.330,0.0100,-0.0900,1.0000
C00481=111.110,15.920,101.590,0.0300,-0.0900,1.0000
C00482=117.580,20.340,102.240,0.0500,-0.0400,1.0000
C00483=120.720,27.280,102.770,0.0300,-0.0000,1.0000
C00484=119.890,35.330,103.300,0.0000,0.0000,1.0000
C00485=117.130,43.660,103.650,0.0000,0.0000,1.0000
C00486=113.690,51.950,103.650,0.0000,0.0000,1.0000
C00487=109.750,59.790,103.300,0.0000,0.0000,1.0000
C00488=104.660,66.070,102.770,0.0200,0.0200,1.0000
C00489=97.520,68.760,102.240,0.0100,0.0600,1.0000
C00490=89.830,67.310,101.590,-0.0400,0.0800,1.0000
C00491=82.560,62.060,100.330,-0.0600,0.0800,1.0000
C00492=74.830,56.040,97.720,-0.0500,0.0700,1.0000
C00493=67.780,50.540,94.220,-0.0400,0.0600,1.0000
C00494=62.260,46.440,90.740,-0.0200,0.0300,1.0000
C00495=58.180,44.800,88.210,-0.0100,-0.3300,0.9400
C00496=54.650,46.780,87.200,-0.3300,-0.4100,0.8500
C00497=52.450,49.090,87.150,-0.4000,-0.3700,0.8400
C00498=50.790,50.790,87.180,-0.3800,-0.3800,0.8400
C00499=49.090,52.450,87.150,-0.3700,-0.4000,0.8400
C00500=46.780,54.650,87.200,-0.4100,-0.3300,0.8500
C00501=44.800,58.180,88.210,-0.3300,-0.0100,0.9400
C00502=46.440,62.260,90.740,0.0300,-0.0200,1.0000
C00503=50.540,67.780,94.220,0.0600,-0.0400,1.0000
C00504=56.040,74.830,97.720,0.0700,-0.0500,1.0000
C00505=62.060,82.560,100.330,0.0800,-0.0600,1.0000
C00506=67.310,89.830,101.590,0.0800,-0.0400,1.0000
C00507=68.760,97.520,102.240,0.0600,0.0100,1.0000
C00508=66.070,104.660,102.770,0.0200,0.0200,1.0000
C00509=59.790,109.750,103.300,0.0000,0.0000,1.0000
C00510=51.950,113.690,103.650,0.0000,0.0000,1.0000
C00511=43.660,117.130,103.650,0.0000,0.0000,1.0000
C00512=35.330,119.890,103.300,0.0000,0.0000,1.0000
C00513=27.280,120.720,102.770,-0.0000,0.0300,1.0000
C00514=20.340,117.580,102.240,-0.0400,0.0500,1.0000
C00515=15.920,111.110,101.590,-0.0900,0.0300,1.0000
C00516=14.500,102.260,100.330,-0.0900,0.0100,1.0000
C00517=13.290,92.540,97.720,-0.0900,0.0100,1.0000
C00518=12.190,83.660,94.220,-0.0700,0.0100,1.0000
C00519=11.190,76.860,90.740,-0.0300,0.0100,1.0000
C00520=9.460,72.820,88.210,0.2300,-0.2400,0.9400
C00521=5.560,71.730,87.200,0.0500,-0.5300,0.8500
C00522=2.380,71.800,87.150,-0.0200,-0.5400,0.8400
C00523=0.000,71.830,87.180,-0.0000,-0.5400,0.8400
C00524=0.000,70.920,88.620,-0.0000,-0.5300,0.8500
C00525=2.300,70.890,88.590,-0.0200,-0.5300,0.8500
C00526=5.420,70.830,88.630,0.0600,-0.5100,0.8600
C00527=9.300,71.960,89.660,0.2200,-0.2200,0.9500
C00528=10.990,76.120,92.260,-0.0300,0.0100,1.0000
C00529=11.980,83.090,95.800,-0.0700,0.0100,1.0000
C00530=13.090,92.160,99.360,-0.0800,0.0100,1.0000
C00531=14.310,102.040,102.000,-0.0900,0.0100,1.0000
C00532=15.730,111.010,103.270,-0.0800,0.0300,1.0000
C00533=20.160,117.560,103.930,-0.0300,0.0400,1.0000
C00534=27.150,120.750,104.470,-0.0000,0.0300,1.0000
C00535=35.250,119.910,105.000,0.0000,0.0000,1.0000
C00536=43.630,117.140,105.350,0.0000,0.0000,1.0000
C00537=51.980,113.680,105.350,0.0000,0.0000,1.0000
C00538=59.870,109.710,105.000,0.0000,0.0000,1.0000
C00539=66.180,104.580,104.470,0.0200,0.0200,1.0000
C00540=68.870,97.380,103.930,0.0500,0.0100,1.0000
C00541=67.370,89.620,103.270,0.0800,-0.0400,1.0000
C00542=62.030,82.270,102.000,0.0700,-0.0500,1.0000
C00543=55.910,74.420,99.360,0.0700,-0.0500,1.0000
C00544=50.280,67.230,95.800,0.0600,-0.0400,1.0000
C00545=46.050,61.590,92.260,0.0300,-0.0200,1.0000
C00546=44.310,57.460,89.660,-0.3100,-0.0000,0.9500
C00547=46.250,53.920,88.630,-0.4000,-0.3200,0.8600
C00548=48.500,51.750,88.590,-0.3600,-0.3900,0.8500
C00549=50.150,50.150,88.620,-0.3800,-0.3800,0.8500
C00550=51.750,48.500,88.590,-0.3900,-0.3600,0.8500
C00551=53.920,46.250,88.630,-0.3200,-0.4000,0.8600
C00552=57.460,44.310,89.670,-0.0000,-0.3100,0.9500
C00553=61.590,46.050,92.260,-0.0200,0.0300,1.0000
C00554=67.230,50.280,95.800,-0.0400,0.0600,1.0000
C00555=74.420,55.910,99.360,-0.0500,0.0700,1.0000
C00556=82.270,62.030,102.000,-0.0500,0.0700,1.0000
C00557=89.620,67.370,103.270,-0.0400,0.0800,1.0000
C00558=97.380,68.870,103.930,0.0100,0.0500,1.0000
C00559=104.580,66.180,104.470,0.0200,0.0200,1.0000
C00560=109.710,59.870,105.000,0.0000,0.0000,1.0000
C00561=113.680,51.980,105.350,0.0000,0.0000,1.0000
C00562=117.140,43.630,105.350,0.0000,0.0000,1.0000
C00563=119.910,35.250,105.000,0.0000,0.0000,1.0000
C00564=120.750,27.150,104.470,0.0300,-0.0000,1.0000
C00565=117.560,20.160,103.930,0.0400,-0.0300,1.0000
C00566=111.010,15.730,103.270,0.0300,-0.0800,1.0000
C00567=102.040,14.310,102.000,0.0100,-0.0900,1.0000
C00568=92.160,13.090,99.360,0.0100,-0.0800,1.0000
C00569=83.090,11.980,95.800,0.0100,-0.0700,1.0000
C00570=76.120,10.990,92.260,0.0100,-0.0300,1.0000
C00571=71.960,9.300,89.660,-0.2200,0.2200,0.9500
C00572=70.830,5.420,88.630,-0.5100,0.0600,0.8600
C00573=70.890,2.300,88.590,-0.5300,-0.0200,0.8500
C00574=70.920,0.000,88.620,-0.5300,-0.0000,0.8500
C00575=70.890,-2.300,88.590,-0.5300,0.0200,0.8500
C00576=70.830,-5.420,88.630,-0.5100,-0.0600,0.8600
C00577=71.960,-9.300,89.670,-0.2200,-0.2200,0.9500
C00578=76.120,-10.990,92.260,0.0100,0.0300,1.0000
C00579=83.090,-11.980,95.800,0.0100,0.0700,1.0000
C00580=92.160,-13.090,99.360,0.0100,0.0800,1.0000
C00581=102.040,-14.310,102.000,0.0100,0.0900,1.0000
C00582=111.010,-15.730,103.270,0.0300,0.0800,1.0000
C00583=117.560,-20.160,103.930,0.0400,0.0300,1.0000
C00584=120.750,-27.150,104.470,0.0300,0.0000,1.0000
C00585=119.910,-35.250,105.000,0.0000,-0.0000,1.0000
C00586=117.140,-43.630,105.350,0.0000,-0.0000,1.0000
C00587=113.680,-51.980,105.350,0.0000,-0.0000,1.0000
C00588=109.710,-59.870,105.000,0.0000,-0.0000,1.0000
C00589=104.580,-66.180,104.470,0.0200,-0.0200,1.0000
C00590=97.380,-68.870,103.930,0.0100,-0.0500,1.0000
C00591=89.620,-67.370,103.270,-0.0400,-0.0800,1.0000
C00592=82.270,-62.030,102.000,-0.0500,-0.0700,1.0000
C00593=74.420,-55.910,99.360,-0.0500,-0.0700,1.0000
C00594=67.230,-50.280,95.800,-0.0400,-0.0600,1.0000
C00595=61.590,-46.050,92.260,-0.0200,-0.0300,1.0000
C00596=57.460,-44.310,89.660,-0.0000,0.3100,0.9500
C00597=53.920,-46.250,88.630,-0.3200,0.4000,0.8600
C00598=51.750,-48.500,88.590,-0.3900,0.3600,0.8500
C00599=50.150,-50.150,88.620,-0.3800,0.3800,0.8500
C00600=48.500,-51.750,88.590,-0.3600,0.3900,0.8500
C00601=46.250,-53.920,88.630,-0.4000,0.3200,0.8600
C00602=44.310,-57.460,89.670,-0.3100,0.0000,0.9500
C00603=46.050,-61.590,92.260,0.0300,0.0200,1.0000
C00604=50.280,-67.230,95.800,0.0600,0.0400,1.0000
C00605=55.910,-74.420,99.360,0.0700,0.0500,1.0000
C00606=62.030,-82.270,102.000,0.0700,0.0500,1.0000
C00607=67.370,-89.620,103.270,0.0800,0.0400,1.0000
C00608=68.870,-97.380,103.930,0.0500,-0.0100,1.0000
C00609=66.180,-104.580,104.470,0.0200,-0.0200,1.0000
C00610=59.870,-109.710,105.000,0.0000,-0.0000,1.0000
C00611=51.980,-113.680,105.350,0.0000,-0.0000,1.0000
C00612=43.630,-117.140,105.350,0.0000,-0.0000,1.0000
C00613=35.250,-119.910,105.000,0.0000,-0.0000,1.0000
C00614=27.150,-120.750,104.470,-0.0000,-0.0300,1.0000
C00615=20.160,-117.560,103.930,-0.0300,-0.0400,1.0000
C00616=15.730,-111.010,103.270,-0.0800,-0.0300,1.0000
C00617=14.310,-102.040,102.000,-0.0900,-0.0100,1.0000
C00618=13.090,-92.160,99.360,-0.0800,-0.0100,1.0000
C00619=11.980,-83.090,95.800,-0.0700,-0.0100,1.0000
C00620=10.990,-76.120,92.260,-0.0300,-0.0100,1.0000
C00621=9.300,-71.960,89.660,0.2200,0.2200,0.9500
C00622=5.420,-70.830,88.630,0.0600,0.5100,0.8600
C00623=2.300,-70.890,88.590,-0.0200,0.5300,0.8500
C00624=0.000,-70.920,88.620,-0.0000,0.5300,0.8500
C00625=0.000,-70.920,88.620,-0.0000,0.5300,0.8500
C00626=-2.300,-70.890,88.590,0.0200,0.5300,0.8500
C00627=-5.420,-70.830,88.630,-0.0600,0.5100,0.8600
C00628=-9.300,-71.960,89.670,-0.2200,0.2200,0.9500
C00629=-10.990,-76.120,92.260,0.0300,-0.0100,1.0000
C00630=-11.980,-83.090,95.800,0.0700,-0.0100,1.0000
C00631=-13.090,-92.160,99.360,0.0800,-0.0100,1.0000
C00632=-14.310,-102.040,102.000,0.0900,-0.0100,1.0000
C00633=-15.730,-111.010,103.270,0.0800,-0.0300,1.0000
C00634=-20.160,-117.560,103.930,0.0300,-0.0400,1.0000
C00635=-27.150,-120.750,104.470,0.0000,-0.0300,1.0000
C00636=-35.250,-119.910,105.000,-0.0000,-0.0000,1.0000
C00637=-43.630,-117.140,105.350,-0.0000,-0.0000,1.0000
C00638=-51.980,-113.680,105.350,-0.0000,-0.0000,1.0000
C00639=-59.870,-109.710,105.000,-0.0000,-0.0000,1.0000
C00640=-66.180,-104.580,104.470,-0.0200,-0.0200,1.0000
C00641=-68.870,-97.380,103.930,-0.0500,-0.0100,1.0000
C00642=-67.370,-89.620,103.270,-0.0800,0.0400,1.0000
C00643=-62.030,-82.270,102.000,-0.0700,0.0500,1.0000
C00644=-55.910,-74.420,99.360,-0.0700,0.0500,1.0000
C00645=-50.280,-67.230,95.800,-0.0600,0.0400,1.0000
C00646=-46.050,-61.590,92.260,-0.0300,0.0200,1.0000
C00647=-44.310,-57.460,89.660,0.3100,0.0000,0.9500
C00648=-46.250,-53.920,88.630,0.4000,0.3200,0.8600
C00649=-48.500,-51.750,88.590,0.3600,0.3900,0.8500
C00650=-50.150,-50.150,88.620,0.3800,0.3800,0.8500
C00651=-51.750,-48.500,88.590,0.3900,0.3600,0.8500
C00652=-53.920,-46.250,88.630,0.3200,0.4000,0.8600
C00653=-57.460,-44.310,89.670,0.0000,0.3100,0.9500
C00654=-61.590,-46.050,92.260,0.0200,-0.0300,1.0000
C00655=-67.230,-50.280,95.800,0.0400,-0.0600,1.0000
C00656=-74.420,-55.910,99.360,0.0500,-0.0700,1.0000
C00657=-82.270,-62.030,102.000,0.0500,-0.0700,1.0000
C00658=-89.620,-67.370,103.270,0.0400,-0.0800,1.0000
C00659=-97.380,-68.870,103.930,-0.0100,-0.0500,1.0000
C00660=-104.580,-66.180,104.470,-0.0200,-0.0200,1.0000
C00661=-109.710,-59.870,105.000,-0.0000,-0.0000,1.0000
C00662=-113.680,-51.980,105.350,-0.0000,-0.0000,1.0000
C00663=-117.140,-43.630,105.350,-0.0000,-0.0000,1.0000
C00664=-119.910,-35.250,105.000,-0.0000,-0.0000,1.0000
C00665=-120.750,-27.150,104.470,-0.0300,0.0000,1.0000
C00666=-117.560,-20.160,103.930,-0.0400,0.0300,1.0000
C00667=-111.010,-15.730,103.270,-0.0300,0.0800,1.0000
C00668=-102.040,-14.310,102.000,-0.0100,0.0900,1.0000
C00669=-92.160,-13.090,99.360,-0.0100,0.0800,1.0000
C00670=-83.090,-11.980,95.800,-0.0100,0.0700,1.0000
C00671=-76.120,-10.990,92.260,-0.0100,0.0300,1.0000
C00672=-71.960,-9.300,89.660,0.2200,-0.2200,0.9500
C00673=-70.830,-5.420,88.630,0.5100,-0.0600,0.8600
C00674=-70.890,-2.300,88.590,0.5300,0.0200,0.8500
C00675=-70.920,0.000,88.620,0.5300,0.0000,0.8500
C00676=-70.890,2.300,88.590,0.5300,-0.0200,0.8500
C00677=-70.830,5.420,88.630,0.5100,0.0600,0.8600
C00678=-71.960,9.300,89.670,0.2200,0.2200,0.9500
C00679=-76.120,10.990,92.260,-0.0100,-0.0300,1.0000
C00680=-83.090,11.980,95.800,-0.0100,-0.0700,1.0000
C00681=-92.160,13.090,99.360,-0.0100,-0.0800,1.0000
C00682=-102.040,14.310,102.000,-0.0100,-0.0900,1.0000
C00683=-111.010,15.730,103.270,-0.0300,-0.0800,1.0000
C00684=-117.560,20.160,103.930,-0.0400,-0.0300,1.0000
C00685=-120.750,27.150,104.470,-0.0300,-0.0000,1.0000
C00686=-119.910,35.250,105.000,-0.0000,0.0000,1.0000
C00687=-117.140,43.630,105.350,-0.0000,0.0000,1.0000
C00688=-113.680,51.980,105.350,-0.0000,0.0000,1.0000
C00689=-109.710,59.870,105.000,-0.0000,0.0000,1.0000
C00690=-104.580,66.180,104.470,-0.0200,0.0200,1.0000
C00691=-97.380,68.870,103.930,-0.0100,0.0500,1.0000
C00692=-89.620,67.370,103.270,0.0400,0.0800,1.0000
C00693=-82.270,62.030,102.000,0.0500,0.0700,1.0000
C00694=-74.420,55.910,99.360,0.0500,0.0700,1.0000
C00695=-67.230,50.280,95.800,0.0400,0.0600,1.0000
C00696=-61.590,46.050,92.260,0.0200,0.0300,1.0000
C00697=-57.460,44.310,89.660,0.0000,-0.3100,0.9500
C00698=-53.920,46.250,88.630,0.3200,-0.4000,0.8600
C00699=-51.750,48.500,88.590,0.3900,-0.3600,0.8500
C00700=-50.150,50.150,88.620,0.3800,-0.3800,0.8500
C00701=-48.500,51.750,88.590,0.3600,-0.3900,0.8500
C00702=-46.250,53.920,88.630,0.4000,-0.3200,0.8600
C00703=-44.310,57.460,89.670,0.3100,-0.0000,0.9500
C00704=-46.050,61.590,92.260,-0.0300,-0.0200,1.0000
C00705=-50.280,67.230,95.800,-0.0600,-0.0400,1.0000
C00706=-55.910,74.420,99.360,-0.0700,-0.0500,1.0000
C00707=-62.030,82.270,102.000,-0.0700,-0.0500,1.0000
C00708=-67.370,89.620,103.270,-0.0800,-0.0400,1.0000
C00709=-68.870,97.380,103.930,-0.0500,0.0100,1.0000
C00710=-66.180,104.580,104.470,-0.0200,0.0200,1.0000
C00711=-59.870,109.710,105.000,-0.0000,0.0000,1.0000
C00712=-51.980,113.680,105.350,-0.0000,0.0000,1.0000
C00713=-43.630,117.140,105.350,-0.0000,0.0000,1.0000
C00714=-35.250,119.910,105.000,-0.0000,0.0000,1.0000
C00715=-27.150,120.750,104.470,0.0000,0.0300,1.0000
C00716=-20.160,117.560,103.930,0.0300,0.0400,1.0000
C00717=-15.730,111.010,103.270,0.0800,0.0300,1.0000
C00718=-14.310,102.040,102.000,0.0900,0.0100,1.0000
C00719=-13.090,92.160,99.360,0.0800,0.0100,1.0000
C00720=-11.980,83.090,95.800,0.0700,0.0100,1.0000
C00721=-10.990,76.120,92.260,0.0300,0.0100,1.0000
C00722=-9.300,71.960,89.670,-0.2200,-0.2200,0.9500
C00723=-5.420,70.830,88.630,-0.0600,-0.5100,0.8600
C00724=-2.300,70.890,88.590,0.0200,-0.5300,0.8500
C00725=0.000,70.920,88.620,-0.0000,-0.5300,0.8500
C00726=0.000,70.020,90.060,-0.0000,-0.5200,0.8500
C00727=-2.220,70.000,90.030,0.0200,-0.5200,0.8500
C00728=-5.290,69.940,90.080,-0.0600,-0.5000,0.8600
C00729=-9.130,71.130,91.140,-0.2100,-0.2100,0.9500
C00730=-10.800,75.400,93.790,0.0400,0.0100,1.0000
C00731=-11.790,82.540,97.400,0.0700,0.0100,1.0000
C00732=-12.900,91.790,101.010,0.0800,0.0100,1.0000
C00733=-14.130,101.830,103.680,0.0800,0.0100,1.0000
C00734=-15.550,110.910,104.960,0.0700,0.0200,1.0000
C00735=-20.000,117.540,105.630,0.0300,0.0400,1.0000
C00736=-27.030,120.770,106.160,0.0000,0.0200,1.0000
C00737=-35.170,119.940,106.700,-0.0000,0.0000,1.0000
C00738=-43.610,117.150,107.050,-0.0000,0.0000,1.0000
C00739=-52.000,113.670,107.050,-0.0000,0.0000,1.0000
C00740=-59.940,109.680,106.700,-0.0000,0.0000,1.0000
C00741=-66.290,104.510,106.160,-0.0200,0.0100,1.0000
C00742=-68.970,97.250,105.630,-0.0500,0.0000,1.0000
C00743=-67.430,89.420,104.960,-0.0700,-0.0400,1.0000
C00744=-62.010,82.000,103.680,-0.0700,-0.0500,1.0000
C00745=-55.780,74.030,101.010,-0.0600,-0.0500,1.0000
C00746=-50.030,66.700,97.400,-0.0500,-0.0400,1.0000
C00747=-45.680,60.950,93.790,-0.0300,-0.0200,1.0000
C00748=-43.840,56.750,91.140,0.3000,0.0000,0.9500
C00749=-45.720,53.200,90.080,0.4000,-0.3100,0.8600
C00750=-47.930,51.060,90.030,0.3500,-0.3800,0.8500
C00751=-49.510,49.510,90.060,0.3700,-0.3700,0.8500
C00752=-51.060,47.930,90.030,0.3800,-0.3500,0.8500
C00753=-53.200,45.720,90.080,0.3100,-0.4000,0.8600
C00754=-56.750,43.840,91.140,-0.0000,-0.3000,0.9500
C00755=-60.950,45.680,93.790,0.0200,0.0300,1.0000
C00756=-66.700,50.030,97.400,0.0400,0.0500,1.0000
C00757=-74.030,55.780,101.010,0.0500,0.0600,1.0000
C00758=-82.000,62.010,103.680,0.0500,0.0700,1.0000
C00759=-89.420,67.430,104.960,0.0400,0.0700,1.0000
C00760=-97.250,68.970,105.630,-0.0000,0.0500,1.0000
C00761=-104.510,66.290,106.160,-0.0100,0.0200,1.0000
C00762=-109.680,59.940,106.700,-0.0000,0.0000,1.0000
C00763=-113.670,52.000,107.050,-0.0000,0.0000,1.0000
C00764=-117.150,43.610,107.050,-0.0000,0.0000,1.0000
C00765=-119.940,35.170,106.700,-0.0000,0.0000,1.0000
C00766=-120.770,27.030,106.160,-0.0200,-0.0000,1.0000
C00767=-117.540,20.000,105.630,-0.0400,-0.0300,1.0000
C00768=-110.910,15.550,104.960,-0.0200,-0.0700,1.0000
C00769=-101.830,14.130,103.680,-0.0100,-0.0800,1.0000
C00770=-91.790,12.900,101.010,-0.0100,-0.0800,1.0000
C00771=-82.540,11.790,97.400,-0.0100,-0.0700,1.0000
C00772=-75.400,10.800,93.790,-0.0100,-0.0400,1.0000
C00773=-71.130,9.130,91.140,0.2100,0.2100,0.9500
C00774=-69.940,5.290,90.080,0.5000,0.0600,0.8600
C00775=-70.000,2.220,90.030,0.5200,-0.0200,0.8500
C00776=-70.020,0.000,90.060,0.5200,0.0000,0.8500
C00777=-70.000,-2.220,90.030,0.5200,0.0200,0.8500
C00778=-69.940,-5.290,90.080,0.5000,-0.0600,0.8600
C00779=-71.130,-9.130,91.140,0.2100,-0.2100,0.9500
C00780=-75.400,-10.800,93.790,-0.0100,0.0400,1.0000
C00781=-82.540,-11.790,97.400,-0.0100,0.0700,1.0000
C00782=-91.790,-12.900,101.010,-0.0100,0.0800,1.0000
C00783=-101.830,-14.130,103.680,-0.0100,0.0800,1.0000
C00784=-110.910,-15.550,104.960,-0.0200,0.0700,1.0000
C00785=-117.540,-20.000,105.630,-0.0400,0.0300,1.0000
C00786=-120.770,-27.030,106.160,-0.0200,0.0000,1.0000
C00787=-119.940,-35.170,106.700,-0.0000,-0.0000,1.0000
C00788=-117.150,-43.610,107.050,-0.0000,-0.0000,1.0000
C00789=-113.670,-52.000,107.050,-0.0000,-0.0000,1.0000
C00790=-109.680,-59.940,106.700,-0.0000,-0.0000,1.0000
C00791=-104.510,-66.290,106.160,-0.0100,-0.0200,1.0000
C00792=-97.250,-68.970,105.630,-0.0000,-0.0500,1.0000
C00793=-89.420,-67.430,104.960,0.0400,-0.0700,1.0000
C00794=-82.000,-62.010,103.680,0.0500,-0.0700,1.0000
C00795=-74.030,-55.780,101.010,0.0500,-0.0600,1.0000
C00796=-66.700,-50.030,97.400,0.0400,-0.0500,1.0000
C00797=-60.950,-45.680,93.790,0.0200,-0.0300,1.0000
C00798=-56.750,-43.840,91.140,-0.0000,0.3000,0.9500
C00799=-53.200,-45.720,90.080,0.3100,0.4000,0.8600
C00800=-51.060,-47.930,90.030,0.3800,0.3500,0.8500
C00801=-49.510,-49.510,90.060,0.3700,0.3700,0.8500
C00802=-47.930,-51.060,90.030,0.3500,0.3800,0.8500
C00803=-45.720,-53.200,90.080,0.4000,0.3100,0.8600
C00804=-43.840,-56.750,91.140,0.3000,-0.0000,0.9500
C00805=-45.680,-60.950,93.790,-0.0300,0.0200,1.0000
C00806=-50.030,-66.700,97.400,-0.0500,0.0400,1.0000
C00807=-55.780,-74.030,101.010,-0.0600,0.0500,1.0000
C00808=-62.010,-82.000,103.680,-0.0700,0.0500,1.0000
C00809=-67.430,-89.420,104.960,-0.0700,0.0400,1.0000
C00810=-68.970,-97.250,105.630,-0.0500,-0.0000,1.0000
C00811=-66.290,-104.510,106.160,-0.0200,-0.0100,1.0000
C00812=-59.940,-109.680,106.700,-0.0000,-0.0000,1.0000
C00813=-52.000,-113.670,107.050,-0.0000,-0.0000,1.0000
C00814=-43.610,-117.150,107.050,-0.0000,-0.0000,1.0000
C00815=-35.170,-119.940,106.700,-0.0000,-0.0000,1.0000
C00816=-27.030,-120.770,106.160,0.0000,-0.0200,1.0000
C00817=-20.000,-117.540,105.630,0.0300,-0.0400,1.0000
C00818=-15.550,-110.910,104.960,0.0700,-0.0200,1.0000
C00819=-14.130,-101.830,103.680,0.0800,-0.0100,1.0000
C00820=-12.900,-91.790,101.010,0.0800,-0.0100,1.0000
C00821=-11.790,-82.540,97.400,0.0700,-0.0100,1.0000
C00822=-10.800,-75.400,93.790,0.0400,-0.0100,1.0000
C00823=-9.130,-71.130,91.140,-0.2100,0.2100,0.9500
C00824=-5.290,-69.940,90.080,-0.0600,0.5000,0.8600
C00825=-2.220,-70.000,90.030,0.0200,0.5200,0.8500
C00826=0.000,-70.020,90.060,-0.0000,0.5200,0.8500
C00827=0.000,-70.020,90.060,-0.0000,0.5200,0.8500
C00828=2.220,-70.000,90.030,-0.0200,0.5200,0.8500
C00829=5.290,-69.940,90.080,0.0600,0.5000,0.8600
C00830=9.130,-71.130,91.140,0.2100,0.2100,0.9500
C00831=10.800,-75.400,93.790,-0.0400,-0.0100,1.0000
C00832=11.790,-82.540,97.400,-0.0700,-0.0100,1.0000
C00833=12.900,-91.790,101.010,-0.0800,-0.0100,1.0000
C00834=14.130,-101.830,103.680,-0.0800,-0.0100,1.0000
C00835=15.550,-110.910,104.960,-0.0700,-0.0200,1.0000
C00836=20.000,-117.540,105.630,-0.0300,-0.0400,1.0000
C00837=27.030,-120.770,106.160,-0.0000,-0.0200,1.0000
C00838=35.170,-119.940,106.700,0.0000,-0.0000,1.0000
C00839=43.610,-117.150,107.050,0.0000,-0.0000,1.0000
C00840=52.000,-113.670,107.050,0.0000,-0.0000,1.0000
C00841=59.940,-109.680,106.700,0.0000,-0.0000,1.0000
C00842=66.290,-104.510,106.160,0.0200,-0.0100,1.0000
C00843=68.970,-97.250,105.630,0.0500,-0.0000,1.0000
C00844=67.430,-89.420,104.960,0.0700,0.0400,1.0000
C00845=62.010,-82.000,103.680,0.0700,0.0500,1.0000
C00846=55.780,-74.030,101.010,0.0600,0.0500,1.0000
C00847=50.030,-66.700,97.400,0.0500,0.0400,1.0000
C00848=45.680,-60.950,93.790,0.0300,0.0200,1.0000
C00849=43.840,-56.750,91.140,-0.3000,-0.0000,0.9500
C00850=45.720,-53.200,90.080,-0.4000,0.3100,0.8600
C00851=47.930,-51.060,90.030,-0.3500,0.3800,0.8500
C00852=49.510,-49.510,90.060,-0.3700,0.3700,0.8500
C00853=51.060,-47.930,90.030,-0.3800,0.3500,0.8500
C00854=53.200,-45.720,90.080,-0.3100,0.4000,0.8600
C00855=56.750,-43.840,91.140,0.0000,0.3000,0.9500
C00856=60.950,-45.680,93.790,-0.0200,-0.0300,1.0000
C00857=66.700,-50.030,97.400,-0.0400,-0.0500,1.0000
C00858=74.030,-55.780,101.010,-0.0500,-0.0600,1.0000
C00859=82.000,-62.010,103.680,-0.0500,-0.0700,1.0000
C00860=89.420,-67.430,104.960,-0.0400,-0.0700,1.0000
C00861=97.250,-68.970,105.630,0.0000,-0.0500,1.0000
C00862=104.510,-66.290,106.160,0.0100,-0.0200,1.0000
C00863=109.680,-59.940,106.700,0.0000,-0.0000,1.0000
C00864=113.670,-52.000,107.050,0.0000,-0.0000,1.0000
C00865=117.150,-43.610,107.050,0.0000,-0.0000,1.0000
C00866=119.940,-35.170,106.700,0.0000,-0.0000,1.0000
C00867=120.770,-27.030,106.160,0.0200,0.0000,1.0000
C00868=117.540,-20.000,105.630,0.0400,0.0300,1.0000
C00869=110.910,-15.550,104.960,0.0200,0.0700,1.0000
C00870=101.830,-14.130,103.680,0.0100,0.0800,1.0000
C00871=91.790,-12.900,101.010,0.0100,0.0800,1.0000
C00872=82.540,-11.790,97.400,0.0100,0.0700,1.0000
C00873=75.400,-10.800,93.790,0.0100,0.0400,1.0000
C00874=71.130,-9.130,91.140,-0.2100,-0.2100,0.9500
C00875=69.940,-5.290,90.080,-0.5000,-0.0600,0.8600
C00876=70.000,-2.220,90.030,-0.5200,0.0200,0.8500
C00877=70.020,0.000,90.060,-0.5200,-0.0000,0.8500
C00878=70.000,2.220,90.030,-0.5200,-0.0200,0.8500
C00879=69.940,5.290,90.080,-0.5000,0.0600,0.8600
C00880=71.130,9.130,91.140,-0.2100,0.2100,0.9500
C00881=75.400,10.800,93.790,0.0100,-0.0400,1.0000
C00882=82.540,11.790,97.400,0.0100,-0.0700,1.0000
C00883=91.790,12.900,101.010,0.0100,-0.0800,1.0000
C00884=101.830,14.130,103.680,0.0100,-0.0800,1.0000
C00885=110.910,15.550,104.960,0.0200,-0.0700,1.0000
C00886=117.540,20.000,105.630,0.0400,-0.0300,1.0000
C00887=120.770,27.030,106.160,0.0200,-0.0000,1.0000
C00888=119.940,35.170,106.700,0.0000,0.0000,1.0000
C00889=117.150,43.610,107.050,0.0000,0.0000,1.0000
C00890=113.670,52.000,107.050,0.0000,0.0000,1.0000
C00891=109.680,59.940,106.700,0.0000,0.0000,1.0000
C00892=104.510,66.290,106.160,0.0100,0.0200,1.0000
C00893=97.250,68.970,105.630,0.0000,0.0500,1.0000
C00894=89.420,67.430,104.960,-0.0400,0.0700,1.0000
C00895=82.000,62.010,103.680,-0.0500,0.0700,1.0000
C00896=74.030,55.780,101.010,-0.0500,0.0600,1.0000
C00897=66.700,50.030,97.400,-0.0400,0.0500,1.0000
C00898=60.950,45.680,93.790,-0.0200,0.0300,1.0000
C00899=56.750,43.840,91.140,0.0000,-0.3000,0.9500
C00900=53.200,45.720,90.080,-0.3100,-0.4000,0.8600
C00901=51.060,47.930,90.030,-0.3800,-0.3500,0.8500
C00902=49.510,49.510,90.060,-0.3700,-0.3700,0.8500
C00903=47.930,51.060,90.030,-0.3500,-0.3800,0.8500
C00904=45.720,53.200,90.080,-0.4000,-0.3100,0.8600
C00905=43.840,56.750,91.140,-0.3000,0.0000,0.9500
C00906=45.680,60.950,93.790,0.0300,-0.0200,1.0000
C00907=50.030,66.700,97.400,0.0500,-0.0400,1.0000
C00908=55.780,74.030,101.010,0.0600,-0.0500,1.0000
C00909=62.010,82.000,103.680,0.0700,-0.0500,1.0000
C00910=67.430,89.420,104.960,0.0700,-0.0400,1.0000
C00911=68.970,97.250,105.630,0.0500,0.0000,1.0000
C00912=66.290,104.510,106.160,0.0200,0.0100,1.0000
C00913=59.940,109.680,106.700,0.0000,0.0000,1.0000
C00914=52.000,113.670,107.050,0.0000,0.0000,1.0000
C00915=43.610,117.150,107.050,0.0000,0.0000,1.0000
C00916=35.170,119.940,106.700,0.0000,0.0000,1.0000
C00917=27.030,120.770,106.160,-0.0000,0.0200,1.0000
C00918=20.000,117.540,105.630,-0.0300,0.0400,1.0000
C00919=15.550,110.910,104.960,-0.0700,0.0200,1.0000
C00920=14.130,101.830,103.680,-0.0800,0.0100,1.0000
C00921=12.900,91.790,101.010,-0.0800,0.0100,1.0000
C00922=11.790,82.540,97.400,-0.0700,0.0100,1.0000
C00923=10.800,75.400,93.790,-0.0400,0.0100,1.0000
C00924=9.130,71.130,91.140,0.2100,-0.2100,0.9500
C00925=5.290,69.940,90.080,0.0600,-0.5000,0.8600
C00926=2.220,70.000,90.030,-0.0200,-0.5200,0.8500
C00927=0.000,70.020,90.060,-0.0000,-0.5200,0.8500
C00928=0.000,69.150,91.520,-0.0000,-0.5100,0.8600
C00929=2.140,69.130,91.490,-0.0200,-0.5100,0.8600
C00930=5.150,69.080,91.540,0.0600,-0.4900,0.8700
C00931=8.970,70.320,92.620,0.2000,-0.2000,0.9600
C00932=10.620,74.710,95.330,-0.0400,0.0100,1.0000
C00933=11.600,82.020,99.010,-0.0600,0.0100,1.0000
C00934=12.730,91.450,102.670,-0.0700,0.0100,1.0000
C00935=13.970,101.630,105.360,-0.0700,0.0100,1.0000
C00936=15.390,110.820,106.650,-0.0700,0.0200,1.0000
C00937=19.850,117.520,107.320,-0.0300,0.0300,1.0000
C00938=26.910,120.790,107.860,-0.0000,0.0200,1.0000
C00939=35.100,119.960,108.400,0.0000,0.0000,1.0000
C00940=43.580,117.150,108.750,0.0000,0.0000,1.0000
C00941=52.020,113.660,108.750,0.0000,0.0000,1.0000
C00942=60.000,109.650,108.400,0.0000,0.0000,1.0000
C00943=66.380,104.440,107.860,0.0200,0.0100,1.0000
C00944=69.060,97.140,107.320,0.0400,0.0000,1.0000
C00945=67.480,89.240,106.650,0.0600,-0.0300,1.0000
C00946=61.990,81.750,105.360,0.0600,-0.0500,1.0000
C00947=55.670,73.660,102.670,0.0600,-0.0400,1.0000
C00948=49.790,66.200,99.010,0.0500,-0.0400,1.0000
C00949=45.320,60.330,95.330,0.0300,-0.0200,1.0000
C00950=43.380,56.060,92.620,-0.2800,0.0100,0.9600
C00951=45.210,52.490,91.540,-0.3900,-0.3000,0.8700
C00952=47.370,50.390,91.490,-0.3400,-0.3700,0.8600
C00953=48.900,48.900,91.520,-0.3600,-0.3600,0.8600
C00954=50.390,47.370,91.490,-0.3700,-0.3400,0.8600
C00955=52.490,45.210,91.540,-0.3000,-0.3900,0.8700
C00956=56.060,43.380,92.620,0.0100,-0.2800,0.9600
C00957=60.330,45.320,95.330,-0.0200,0.0300,1.0000
C00958=66.200,49.790,99.010,-0.0400,0.0500,1.0000
C00959=73.660,55.670,102.670,-0.0400,0.0600,1.0000
C00960=81.750,61.990,105.360,-0.0500,0.0600,1.0000
C00961=89.240,67.480,106.650,-0.0300,0.0600,1.0000
C00962=97.140,69.060,107.320,0.0000,0.0400,1.0000
C00963=104.440,66.380,107.860,0.0100,0.0200,1.0000
C00964=109.650,60.000,108.400,0.0000,0.0000,1.0000
C00965=113.660,52.020,108.750,0.0000,0.0000,1.0000
C00966=117.150,43.580,108.750,0.0000,0.0000,1.0000
C00967=119.960,35.100,108.400,0.0000,0.0000,1.0000
C00968=120.790,26.910,107.860,0.0200,-0.0000,1.0000
C00969=117.520,19.850,107.320,0.0300,-0.0300,1.0000
C00970=110.820,15.390,106.650,0.0200,-0.0700,1.0000
C00971=101.630,13.970,105.360,0.0100,-0.0700,1.0000
C00972=91.450,12.730,102.670,0.0100,-0.0700,1.0000
C00973=82.020,11.600,99.010,0.0100,-0.0600,1.0000
C00974=74.710,10.620,95.330,0.0100,-0.0400,1.0000
C00975=70.320,8.970,92.620,-0.2000,0.2000,0.9600
C00976=69.080,5.150,91.540,-0.4900,0.0600,0.8700
C00977=69.130,2.140,91.490,-0.5100,-0.0200,0.8600
C00978=69.150,0.000,91.520,-0.5100,-0.0000,0.8600
C00979=69.130,-2.140,91.490,-0.5100,0.0200,0.8600
C00980=69.080,-5.150,91.540,-0.4900,-0.0600,0.8700
C00981=70.320,-8.970,92.620,-0.2000,-0.2000,0.9600
C00982=74.710,-10.620,95.330,0.0100,0.0400,1.0000
C00983=82.020,-11.600,99.010,0.0100,0.0600,1.0000
C00984=91.450,-12.730,102.670,0.0100,0.0700,1.0000
C00985=101.630,-13.970,105.360,0.0100,0.0700,1.0000
C00986=110.820,-15.390,106.650,0.0200,0.0700,1.0000
C00987=117.520,-19.850,107.320,0.0300,0.0300,1.0000
C00988=120.790,-26.910,107.860,0.0200,0.0000,1.0000
C00989=119.960,-35.100,108.400,0.0000,-0.0000,1.0000
C00990=117.150,-43.580,108.750,0.0000,-0.0000,1.0000
C00991=113.660,-52.020,108.750,0.0000,-0.0000,1.0000
C00992=109.650,-60.000,108.400,0.0000,-0.0000,1.0000
C00993=104.440,-66.380,107.860,0.0100,-0.0200,1.0000
C00994=97.140,-69.060,107.320,0.0000,-0.0400,1.0000
C00995=89.240,-67.480,106.650,-0.0300,-0.0600,1.0000
C00996=81.750,-61.990,105.360,-0.0500,-0.0600,1.0000
C00997=73.660,-55.670,102.670,-0.0400,-0.0600,1.0000
C00998=66.200,-49.790,99.010,-0.0400,-0.0500,1.0000
C00999=60.330,-45.320,95.330,-0.0200,-0.0300,1.0000
C01000=56.060,-43.380,92.620,0.0100,0.2800,0.9600
C01001=52.490,-45.210,91.540,-0.3000,0.3900,0.8700
C01002=50.390,-47.370,91.490,-0.3700,0.3400,0.8600
C01003=48.900,-48.900,91.520,-0.3600,0.3600,0.8600
C01004=47.370,-50.390,91.490,-0.3400,0.3700,0.8600
C01005=45.210,-52.490,91.540,-0.3900,0.3000,0.8700
C01006=43.380,-56.060,92.620,-0.2800,-0.0100,0.9600
C01007=45.320,-60.330,95.330,0.0300,0.0200,1.0000
C01008=49.790,-66.200,99.010,0.0500,0.0400,1.0000
C01009=55.670,-73.660,102.670,0.0600,0.0400,1.0000
C01010=61.990,-81.750,105.360,0.0600,0.0500,1.0000
C01011=67.480,-89.240,106.650,0.0600,0.0300,1.0000
C01012=69.060,-97.140,107.320,0.0400,-0.0000,1.0000
C01013=66.380,-104.440,107.860,0.0200,-0.0100,1.0000
C01014=60.000,-109.650,108.400,0.0000,-0.0000,1.0000
C01015=52.020,-113.660,108.750,0.0000,-0.0000,1.0000
C01016=43.580,-117.150,108.750,0.0000,-0.0000,1.0000
C01017=35.100,-119.960,108.400,0.0000,-0.0000,1.0000
C01018=26.910,-120.790,107.860,-0.0000,-0.0200,1.0000
C01019=19.850,-117.520,107.320,-0.0300,-0.0300,1.0000
C01020=15.390,-110.820,106.650,-0.0700,-0.0200,1.0000
C01021=13.970,-101.630,105.360,-0.0700,-0.0100,1.0000
C01022=12.730,-91.450,102.670,-0.0700,-0.0100,1.0000
C01023=11.600,-82.020,99.010,-0.0600,-0.0100,1.0000
C01024=10.620,-74.710,95.330,-0.0400,-0.0100,1.0000
C01025=8.970,-70.320,92.620,0.2000,0.2000,0.9600
C01026=5.150,-69.080,91.540,0.0600,0.4900,0.8700
C01027=2.140,-69.130,91.490,-0.0200,0.5100,0.8600
C01028=0.000,-69.150,91.520,-0.0000,0.5100,0.8600
C01029=0.000,-69.150,91.520,-0.0000,0.5100,0.8600
C01030=-2.140,-69.130,91.490,0.0200,0.5100,0.8600
C01031=-5.150,-69.080,91.540,-0.0600,0.4900,0.8700
C01032=-8.970,-70.320,92.620,-0.2000,0.2000,0.9600
C01033=-10.620,-74.710,95.330,0.0400,-0.0100,1.0000
C01034=-11.600,-82.020,99.010,0.0600,-0.0100,1.0000
C01035=-12.730,-91.450,102.670,0.0700,-0.0100,1.0000
C01036=-13.970,-101.630,105.360,0.0700,-0.0100,1.0000
C01037=-15.390,-110.820,106.650,0.0700,-0.0200,1.0000
C01038=-19.850,-117.520,107.320,0.0300,-0.0300,1.0000
C01039=-26.910,-120.790,107.860,0.0000,-0.0200,1.0000
C01040=-35.100,-119.960,108.400,-0.0000,-0.0000,1.0000
C01041=-43.580,-117.150,108.750,-0.0000,-0.0000,1.0000
C01042=-52.020,-113.660,108.750,-0.0000,-0.0000,1.0000
C01043=-60.000,-109.650,108.400,-0.0000,-0.0000,1.0000
C01044=-66.380,-104.440,107.860,-0.0200,-0.0100,1.0000
C01045=-69.060,-97.140,107.320,-0.0400,-0.0000,1.0000
C01046=-67.480,-89.240,106.650,-0.0600,0.0300,1.0000
C01047=-61.990,-81.750,105.360,-0.0600,0.0500,1.0000
C01048=-55.670,-73.660,102.670,-0.0600,0.0400,1.0000
C01049=-49.790,-66.200,99.010,-0.0500,0.0400,1.0000
C01050=-45.320,-60.330,95.330,-0.0300,0.0200,1.0000
C01051=-43.380,-56.060,92.620,0.2800,-0.0100,0.9600
C01052=-45.210,-52.490,91.540,0.3900,0.3000,0.8700
C01053=-47.370,-50.390,91.490,0.3400,0.3700,0.8600
C01054=-48.900,-48.900,91.520,0.3600,0.3600,0.8600
C01055=-50.390,-47.370,91.490,0.3700,0.3400,0.8600
C01056=-52.490,-45.210,91.540,0.3000,0.3900,0.8700
C01057=-56.060,-43.380,92.620,-0.0100,0.2800,0.9600
C01058=-60.330,-45.320,95.330,0.0200,-0.0300,1.0000
C01059=-66.200,-49.790,99.010,0.0400,-0.0500,1.0000
C01060=-73.660,-55.670,102.670,0.0400,-0.0600,1.0000
C01061=-81.750,-61.990,105.360,0.0500,-0.0600,1.0000
C01062=-89.240,-67.480,106.650,0.0300,-0.0600,1.0000
C01063=-97.140,-69.060,107.320,-0.0000,-0.0400,1.0000
C01064=-104.440,-66.380,107.860,-0.0100,-0.0200,1.0000
C01065=-109.650,-60.000,108.400,-0.0000,-0.0000,1.0000
C01066=-113.660,-52.020,108.750,-0.0000,-0.0000,1.0000
C01067=-117.150,-43.580,108.750,-0.0000,-0.0000,1.0000
C01068=-119.960,-35.100,108.400,-0.0000,-0.0000,1.0000
C01069=-120.790,-26.910,107.860,-0.0200,0.0000,1.0000
C01070=-117.520,-19.850,107.320,-0.0300,0.0300,1.0000
C01071=-110.820,-15.390,106.650,-0.0200,0.0700,1.0000
C01072=-101.630,-13.970,105.360,-0.0100,0.0700,1.0000
C01073=-91.450,-12.730,102.670,-0.0100,0.0700,1.0000
C01074=-82.020,-11.600,99.010,-0.0100,0.0600,1.0000
C01075=-74.710,-10.620,95.330,-0.0100,0.0400,1.0000
C01076=-70.320,-8.970,92.620,0.2000,-0.2000,0.9600
C01077=-69.080,-5.150,91.540,0.4900,-0.0600,0.8700
C01078=-69.130,-2.140,91.490,0.5100,0.0200,0.8600
C01079=-69.150,0.000,91.520,0.5100,0.0000,0.8600
C01080=-69.130,2.140,91.490,0.5100,-0.0200,0.8600
C01081=-69.080,5.150,91.540,0.4900,0.0600,0.8700
C01082=-70.320,8.970,92.620,0.2000,0.2000,0.9600
C01083=-74.710,10.620,95.330,-0.0100,-0.0400,1.0000
C01084=-82.020,11.600,99.010,-0.0100,-0.0600,1.0000
C01085=-91.450,12.730,102.670,-0.0100,-0.0700,1.0000
C01086=-101.630,13.970,105.360,-0.0100,-0.0700,1.0000
C01087=-110.820,15.390,106.650,-0.0200,-0.0700,1.0000
C01088=-117.520,19.850,107.320,-0.0300,-0.0300,1.0000
C01089=-120.790,26.910,107.860,-0.0200,-0.0000,1.0000
C01090=-119.960,35.100,108.400,-0.0000,0.0000,1.0000
C01091=-117.150,43.580,108.750,-0.0000,0.0000,1.0000
C01092=-113.660,52.020,108.750,-0.0000,0.0000,1.0000
C01093=-109.650,60.000,108.400,-0.0000,0.0000,1.0000
C01094=-104.440,66.380,107.860,-0.0100,0.0200,1.0000
C01095=-97.140,69.060,107.320,-0.0000,0.0400,1.0000
C01096=-89.240,67.480,106.650,0.0300,0.0600,1.0000
C01097=-81.750,61.990,105.360,0.0500,0.0600,1.0000
C01098=-73.660,55.670,102.670,0.0400,0.0600,1.0000
C01099=-66.200,49.790,99.010,0.0400,0.0500,1.0000
C01100=-60.330,45.320,95.330,0.0200,0.0300,1.0000
C01101=-56.060,43.380,92.620,-0.0100,-0.2800,0.9600
C01102=-52.490,45.210,91.540,0.3000,-0.3900,0.8700
C01103=-50.390,47.370,91.490,0.3700,-0.3400,0.8600
C01104=-48.900,48.900,91.520,0.3600,-0.3600,0.8600
C01105=-47.370,50.390,91.490,0.3400,-0.3700,0.8600
C01106=-45.210,52.490,91.540,0.3900,-0.3000,0.8700
C01107=-43.380,56.060,92.620,0.2800,0.0100,0.9600
C01108=-45.320,60.330,95.330,-0.0300,-0.0200,1.0000
C01109=-49.790,66.200,99.010,-0.0500,-0.0400,1.0000
C01110=-55.670,73.660,102.670,-0.0600,-0.0400,1.0000
C01111=-61.990,81.750,105.360,-0.0600,-0.0500,1.0000
C01112=-67.480,89.240,106.650,-0.0600,-0.0300,1.0000
C01113=-69.060,97.140,107.320,-0.0400,0.0000,1.0000
C01114=-66.380,104.440,107.860,-0.0200,0.0100,1.0000
C01115=-60.000,109.650,108.400,-0.0000,0.0000,1.0000
C01116=-52.020,113.660,108.750,-0.0000,0.0000,1.0000
C01117=-43.580,117.150,108.750,-0.0000,0.0000,1.0000
C01118=-35.100,119.960,108.400,-0.0000,0.0000,1.0000
C01119=-26.910,120.790,107.860,0.0000,0.0200,1.0000
C01120=-19.850,117.520,107.320,0.0300,0.0300,1.0000
C01121=-15.390,110.820,106.650,0.0700,0.0200,1.0000
C01122=-13.970,101.630,105.360,0.0700,0.0100,1.0000
C01123=-12.730,91.450,102.670,0.0700,0.0100,1.0000
C01124=-11.600,82.020,99.010,0.0600,0.0100,1.0000
C01125=-10.620,74.710,95.330,0.0400,0.0100,1.0000
C01126=-8.970,70.320,92.620,-0.2000,-0.2000,0.9600
C01127=-5.150,69.080,91.540,-0.0600,-0.4900,0.8700
C01128=-2.140,69.130,91.490,0.0200,-0.5100,0.8600
C01129=0.000,69.150,91.520,-0.0000,-0.5100,0.8600
C01130=0.000,68.300,92.990,-0.0000,-0.4900,0.8700
C01131=-2.060,68.280,92.960,0.0200,-0.4900,0.8700
C01132=-5.020,68.250,93.010,-0.0600,-0.4700,0.8800
C01133=-8.820,69.530,94.120,-0.2000,-0.1800,0.9600
C01134=-10.440,74.040,96.890,0.0400,0.0100,1.0000
C01135=-11.420,81.530,100.630,0.0600,0.0100,1.0000
C01136=-12.570,91.130,104.330,0.0700,0.0100,1.0000
C01137=-13.830,101.460,107.040,0.0700,0.0100,1.0000
C01138=-15.240,110.740,108.340,0.0600,0.0200,1.0000
C01139=-19.720,117.510,109.010,0.0300,0.0300,1.0000
C01140=-26.820,120.810,109.560,0.0000,0.0200,1.0000
C01141=-35.040,119.980,110.100,-0.0000,0.0000,1.0000
C01142=-43.560,117.160,110.450,-0.0000,0.0000,1.0000
C01143=-52.040,113.650,110.450,-0.0000,0.0000,1.0000
C01144=-60.060,109.620,110.100,-0.0000,0.0000,1.0000
C01145=-66.460,104.390,109.560,-0.0200,0.0100,1.0000
C01146=-69.140,97.040,109.010,-0.0400,0.0000,1.0000
C01147=-67.530,89.090,108.340,-0.0600,-0.0300,1.0000
C01148=-61.970,81.520,107.040,-0.0500,-0.0400,1.0000
C01149=-55.560,73.330,104.330,-0.0500,-0.0400,1.0000
C01150=-49.570,65.730,100.630,-0.0500,-0.0400,1.0000
C01151=-44.970,59.740,96.890,-0.0300,-0.0200,1.0000
C01152=-42.930,55.400,94.120,0.2700,0.0100,0.9600
C01153=-44.710,51.810,93.010,0.3800,-0.2900,0.8800
C01154=-46.830,49.740,92.960,0.3400,-0.3600,0.8700
C01155=-48.300,48.300,92.990,0.3500,-0.3500,0.8700
C01156=-49.740,46.830,92.960,0.3600,-0.3400,0.8700
C01157=-51.810,44.710,93.010,0.2900,-0.3800,0.8800
C01158=-55.400,42.930,94.120,-0.0100,-0.2700,0.9600
C01159=-59.740,44.970,96.890,0.0200,0.0300,1.0000
C01160=-65.730,49.570,100.630,0.0400,0.0500,1.0000
C01161=-73.330,55.560,104.330,0.0400,0.0500,1.0000
C01162=-81.520,61.970,107.040,0.0400,0.0500,1.0000
C01163=-89.090,67.530,108.340,0.0300,0.0600,1.0000
C01164=-97.040,69.140,109.010,-0.0000,0.0400,1.0000
C01165=-104.390,66.460,109.560,-0.0100,0.0200,1.0000
C01166=-109.620,60.060,110.100,-0.0000,0.0000,1.0000
C01167=-113.650,52.040,110.450,-0.0000,0.0000,1.0000
C01168=-117.160,43.560,110.450,-0.0000,0.0000,1.0000
C01169=-119.980,35.040,110.100,-0.0000,0.0000,1.0000
C01170=-120.810,26.820,109.560,-0.0200,-0.0000,1.0000
C01171=-117.510,19.720,109.010,-0.0300,-0.0300,1.0000
C01172=-110.740,15.240,108.340,-0.0200,-0.0600,1.0000
C01173=-101.460,13.830,107.040,-0.0100,-0.0700,1.0000
C01174=-91.130,12.570,104.330,-0.0100,-0.0700,1.0000
C01175=-81.530,11.420,100.630,-0.0100,-0.0600,1.0000
C01176=-74.040,10.440,96.890,-0.0100,-0.0400,1.0000
C01177=-69.530,8.820,94.120,0.1800,0.2000,0.9600
C01178=-68.250,5.020,93.010,0.4700,0.0600,0.8800
C01179=-68.280,2.060,92.960,0.4900,-0.0200,0.8700
C01180=-68.300,0.000,92.990,0.4900,0.0000,0.8700
C01181=-68.280,-2.060,92.960,0.4900,0.0200,0.8700
C01182=-68.250,-5.020,93.010,0.4700,-0.0600,0.8800
C01183=-69.530,-8.820,94.120,0.1800,-0.2000,0.9600
C01184=-74.040,-10.440,96.890,-0.0100,0.0400,1.0000
C01185=-81.530,-11.420,100.630,-0.0100,0.0600,1.0000
C01186=-91.130,-12.570,104.330,-0.0100,0.0700,1.0000
C01187=-101.460,-13.830,107.040,-0.0100,0.0700,1.0000
C01188=-110.740,-15.240,108.340,-0.0200,0.0600,1.0000
C01189=-117.510,-19.720,109.010,-0.0300,0.0300,1.0000
C01190=-120.810,-26.820,109.560,-0.0200,0.0000,1.0000
C01191=-119.980,-35.040,110.100,-0.0000,-0.0000,1.0000
C01192=-117.160,-43.560,110.450,-0.0000,-0.0000,1.0000
C01193=-113.650,-52.040,110.450,-0.0000,-0.0000,1.0000
C01194=-109.620,-60.060,110.100,-0.0000,-0.0000,1.0000
C01195=-104.390,-66.460,109.560,-0.0100,-0.0200,1.0000
C01196=-97.040,-69.140,109.010,-0.0000,-0.0400,1.0000
C01197=-89.090,-67.530,108.340,0.0300,-0.0600,1.0000
C01198=-81.520,-61.970,107.040,0.0400,-0.0500,1.0000
C01199=-73.330,-55.560,104.330,0.0400,-0.0500,1.0000
C01200=-65.730,-49.570,100.630,0.0400,-0.0500,1.0000
C01201=-59.740,-44.970,96.890,0.0200,-0.0300,1.0000
C01202=-55.400,-42.930,94.120,-0.0100,0.2700,0.9600
C01203=-51.810,-44.710,93.010,0.2900,0.3800,0.8800
C01204=-49.740,-46.830,92.960,0.3600,0.3400,0.8700
C01205=-48.300,-48.300,92.990,0.3500,0.3500,0.8700
C01206=-46.830,-49.740,92.960,0.3400,0.3600,0.8700
C01207=-44.710,-51.810,93.010,0.3800,0.2900,0.8800
C01208=-42.930,-55.400,94.120,0.2700,-0.0100,0.9600
C01209=-44.970,-59.740,96.890,-0.0300,0.0200,1.0000
C01210=-49.570,-65.730,100.630,-0.0500,0.0400,1.0000
C01211=-55.560,-73.330,104.330,-0.0500,0.0400,1.0000
C01212=-61.970,-81.520,107.040,-0.0500,0.0400,1.0000
C01213=-67.530,-89.090,108.340,-0.0600,0.0300,1.0000
C01214=-69.140,-97.040,109.010,-0.0400,-0.0000,1.0000
C01215=-66.460,-104.390,109.560,-0.0200,-0.0100,1.0000
C01216=-60.060,-109.620,110.100,-0.0000,-0.0000,1.0000
C01217=-52.040,-113.650,110.450,-0.0000,-0.0000,1.0000
C01218=-43.560,-117.160,110.450,-0.0000,-0.0000,1.0000
C01219=-35.040,-119.980,110.100,-0.0000,-0.0000,1.0000
C01220=-26.820,-120.810,109.560,0.0000,-0.0200,1.0000
C01221=-19.720,-117.510,109.010,0.0300,-0.0300,1.0000
C01222=-15.240,-110.740,108.340,0.0600,-0.0200,1.0000
C01223=-13.830,-101.460,107.040,0.0700,-0.0100,1.0000
C01224=-12.570,-91.130,104.330,0.0700,-0.0100,1.0000
C01225=-11.420,-81.530,100.630,0.0600,-0.0100,1.0000
C01226=-10.440,-74.040,96.890,0.0400,-0.0100,1.0000
C01227=-8.820,-69.530,94.120,-0.2000,0.1800,0.9600
C01228=-5.020,-68.250,93.010,-0.0600,0.4700,0.8800
C01229=-2.060,-68.280,92.960,0.0200,0.4900,0.8700
C01230=0.000,-68.300,92.990,-0.0000,0.4900,0.8700
C01231=0.000,-68.300,92.990,-0.0000,0.4900,0.8700
C01232=2.060,-68.280,92.960,-0.0200,0.4900,0.8700
C01233=5.020,-68.250,93.010,0.0600,0.4700,0.8800
C01234=8.820,-69.530,94.120,0.2000,0.1800,0.9600
C01235=10.440,-74.040,96.890,-0.0400,-0.0100,1.0000
C01236=11.420,-81.530,100.630,-0.0600,-0.0100,1.0000
C01237=12.570,-91.130,104.330,-0.0700,-0.0100,1.0000
C01238=13.830,-101.460,107.040,-0.0700,-0.0100,1.0000
C01239=15.240,-110.740,108.340,-0.0600,-0.0200,1.0000
C01240=19.720,-117.510,109.010,-0.0300,-0.0300,1.0000
C01241=26.820,-120.810,109.560,-0.0000,-0.0200,1.0000
C01242=35.040,-119.980,110.100,0.0000,-0.0000,1.0000
C01243=43.560,-117.160,110.450,0.0000,-0.0000,1.0000
C01244=52.040,-113.650,110.450,0.0000,-0.0000,1.0000
C01245=60.060,-109.620,110.100,0.0000,-0.0000,1.0000
C01246=66.460,-104.390,109.560,0.0200,-0.0100,1.0000
C01247=69.140,-97.040,109.010,0.0400,-0.0000,1.0000
C01248=67.530,-89.090,108.340,0.0600,0.0300,1.0000
C01249=61.970,-81.520,107.040,0.0500,0.0400,1.0000
C01250=55.560,-73.330,104.330,0.0500,0.0400,1.0000
C01251=49.570,-65.730,100.630,0.0500,0.0400,1.0000
C01252=44.970,-59.740,96.890,0.0300,0.0200,1.0000
C01253=42.930,-55.400,94.120,-0.2700,-0.0100,0.9600
C01254=44.710,-51.810,93.010,-0.3800,0.2900,0.8800
C01255=46.830,-49.740,92.960,-0.3400,0.3600,0.8700
C01256=48.300,-48.300,92.990,-0.3500,0.3500,0.8700
C01257=49.740,-46.830,92.960,-0.3600,0.3400,0.8700
C01258=51.810,-44.710,93.010,-0.2900,0.3800,0.8800
C01259=55.400,-42.930,94.120,0.0100,0.2700,0.9600
C01260=59.740,-44.970,96.890,-0.0200,-0.0300,1.0000
C01261=65.730,-49.570,100.630,-0.0400,-0.0500,1.0000
C01262=73.330,-55.560,104.330,-0.0400,-0.0500,1.0000
C01263=81.520,-61.970,107.040,-0.0400,-0.0500,1.0000
C01264=89.090,-67.530,108.340,-0.0300,-0.0600,1.0000
C01265=97.040,-69.140,109.010,0.0000,-0.0400,1.0000
C01266=104.390,-66.460,109.560,0.0100,-0.0200,1.0000
C01267=109.620,-60.060,110.100,0.0000,-0.0000,1.0000
C01268=113.650,-52.040,110.450,0.0000,-0.0000,1.0000
C01269=117.160,-43.560,110.450,0.0000,-0.0000,1.0000
C01270=119.980,-35.040,110.100,0.0000,-0.0000,1.0000
C01271=120.810,-26.820,109.560,0.0200,0.0000,1.0000
C01272=117.510,-19.720,109.010,0.0300,0.0300,1.0000
C01273=110.740,-15.240,108.340,0.0200,0.0600,1.0000
C01274=101.460,-13.830,107.040,0.0100,0.0700,1.0000
C01275=91.130,-12.570,104.330,0.0100,0.0700,1.0000
C01276=81.530,-11.420,100.630,0.0100,0.0600,1.0000
C01277=74.040,-10.440,96.890,0.0100,0.0400,1.0000
C01278=69.530,-8.820,94.120,-0.1800,-0.2000,0.9600
C01279=68.250,-5.020,93.010,-0.4700,-0.0600,0.8800
C01280=68.280,-2.060,92.960,-0.4900,0.0200,0.8700
C01281=68.300,0.000,92.990,-0.4900,-0.0000,0.8700
C01282=68.280,2.060,92.960,-0.4900,-0.0200,0.8700
C01283=68.250,5.020,93.010,-0.4700,0.0600,0.8800
C01284=69.530,8.820,94.120,-0.1800,0.2000,0.9600
C01285=74.040,10.440,96.890,0.0100,-0.0400,1.0000
C01286=81.530,11.420,100.630,0.0100,-0.0600,1.0000
C01287=91.130,12.570,104.330,0.0100,-0.0700,1.0000
C01288=101.460,13.830,107.040,0.0100,-0.0700,1.0000
C01289=110.740,15.240,108.340,0.0200,-0.0600,1.0000
C01290=117.510,19.720,109.010,0.0300,-0.0300,1.0000
C01291=120.810,26.820,109.560,0.0200,-0.0000,1.0000
C01292=119.980,35.040,110.100,0.0000,0.0000,1.0000
C01293=117.160,43.560,110.450,0.0000,0.0000,1.0000
C01294=113.650,52.040,110.450,0.0000,0.0000,1.0000
C01295=109.620,60.060,110.100,0.0000,0.0000,1.0000
C01296=104.390,66.460,109.560,0.0100,0.0200,1.0000
C01297=97.040,69.140,109.010,0.0000,0.0400,1.0000
C01298=89.090,67.530,108.340,-0.0300,0.0600,1.0000
C01299=81.520,61.970,107.040,-0.0400,0.0500,1.0000
C01300=73.330,55.560,104.330,-0.0400,0.0500,1.0000
C01301=65.730,49.570,100.630,-0.0400,0.0500,1.0000
C01302=59.740,44.970,96.890,-0.0200,0.0300,1.0000
C01303=55.400,42.930,94.120,0.0100,-0.2700,0.9600
C01304=51.810,44.710,93.010,-0.2900,-0.3800,0.8800
C01305=49.740,46.830,92.960,-0.3600,-0.3400,0.8700
C01306=48.300,48.300,92.990,-0.3500,-0.3500,0.8700
C01307=46.830,49.740,92.960,-0.3400,-0.3600,0.8700
C01308=44.710,51.810,93.010,-0.3800,-0.2900,0.8800
C01309=42.930,55.400,94.120,-0.2700,0.0100,0.9600
C01310=44.970,59.740,96.890,0.0300,-0.0200,1.0000
C01311=49.570,65.730,100.630,0.0500,-0.0400,1.0000
C01312=55.560,73.330,104.330,0.0500,-0.0400,1.0000
C01313=61.970,81.520,107.040,0.0500,-0.0400,1.0000
C01314=67.530,89.090,108.340,0.0600,-0.0300,1.0000
C01315=69.140,97.040,109.010,0.0400,0.0000,1.0000
C01316=66.460,104.390,109.560,0.0200,0.0100,1.0000
C01317=60.060,109.620,110.100,0.0000,0.0000,1.0000
C01318=52.040,113.650,110.450,0.0000,0.0000,1.0000
C01319=43.560,117.160,110.450,0.0000,0.0000,1.0000
C01320=35.040,119.980,110.100,0.0000,0.0000,1.0000
C01321=26.820,120.810,109.560,-0.0000,0.0200,1.0000
C01322=19.720,117.510,109.010,-0.0300,0.0300,1.0000
C01323=15.240,110.740,108.340,-0.0600,0.0200,1.0000
C01324=13.830,101.460,107.040,-0.0700,0.0100,1.0000
C01325=12.570,91.130,104.330,-0.0700,0.0100,1.0000
C01326=11.420,81.530,100.630,-0.0600,0.0100,1.0000
C01327=10.440,74.040,96.890,-0.0400,0.0100,1.0000
C01328=8.820,69.530,94.120,0.2000,-0.1800,0.9600
C01329=5.020,68.250,93.010,0.0600,-0.4700,0.8800
C01330=2.060,68.280,92.960,-0.0200,-0.4900,0.8700
C01331=0.000,68.300,92.990,-0.0000,-0.4900,0.8700
C01332=0.000,67.480,94.480,-0.0000,-0.4800,0.8800
C01333=1.980,67.460,94.450,-0.0200,-0.4800,0.8800
C01334=4.900,67.430,94.500,0.0600,-0.4600,0.8900
C01335=8.660,68.760,95.630,0.1900,-0.1700,0.9700
C01336=10.270,73.410,98.450,-0.0400,0.0100,1.0000
C01337=11.260,81.060,102.250,-0.0600,0.0100,1.0000
C01338=12.420,90.850,106.000,-0.0600,0.0100,1.0000
C01339=13.690,101.300,108.730,-0.0600,0.0100,1.0000
C01340=15.110,110.670,110.040,-0.0500,0.0200,1.0000
C01341=19.610,117.490,110.710,-0.0200,0.0300,1.0000
C01342=26.730,120.820,111.250,-0.0000,0.0200,1.0000
C01343=34.990,120.000,111.800,0.0000,0.0000,1.0000
C01344=43.550,117.170,112.150,0.0000,0.0000,1.0000
C01345=52.060,113.640,112.150,0.0000,0.0000,1.0000
C01346=60.110,109.590,111.800,0.0000,0.0000,1.0000
C01347=66.530,104.340,111.250,0.0100,0.0100,1.0000
C01348=69.210,96.950,110.710,0.0300,0.0000,1.0000
C01349=67.570,88.950,110.040,0.0500,-0.0300,1.0000
C01350=61.950,81.310,108.730,0.0500,-0.0400,1.0000
C01351=55.460,73.020,106.000,0.0500,-0.0400,1.0000
C01352=49.360,65.280,102.250,0.0500,-0.0300,1.0000
C01353=44.640,59.170,98.450,0.0300,-0.0200,1.0000
C01354=42.500,54.750,95.630,-0.2500,0.0100,0.9700
C01355=44.220,51.140,94.500,-0.3700,-0.2800,0.8900
C01356=46.300,49.110,94.450,-0.3200,-0.3500,0.8800
C01357=47.720,47.720,94.480,-0.3400,-0.3400,0.8800
C01358=49.110,46.300,94.450,-0.3500,-0.3200,0.8800
C01359=51.140,44.220,94.500,-0.2800,-0.3700,0.8900
C01360=54.750,42.500,95.630,0.0100,-0.2500,0.9700
C01361=59.170,44.640,98.450,-0.0200,0.0300,1.0000
C01362=65.280,49.360,102.250,-0.0300,0.0500,1.0000
C01363=73.020,55.460,106.000,-0.0400,0.0500,1.0000
C01364=81.310,61.950,108.730,-0.0400,0.0500,1.0000
C01365=88.950,67.570,110.040,-0.0300,0.0500,1.0000
C01366=96.950,69.210,110.710,0.0000,0.0300,1.0000
C01367=104.340,66.530,111.250,0.0100,0.0100,1.0000
C01368=109.590,60.110,111.800,0.0000,0.0000,1.0000
C01369=113.640,52.060,112.150,0.0000,0.0000,1.0000
C01370=117.170,43.550,112.150,0.0000,0.0000,1.0000
C01371=120.000,34.990,111.800,0.0000,0.0000,1.0000
C01372=120.820,26.730,111.250,0.0200,-0.0000,1.0000
C01373=117.490,19.610,110.710,0.0300,-0.0200,1.0000
C01374=110.670,15.110,110.040,0.0200,-0.0500,1.0000
C01375=101.300,13.690,108.730,0.0100,-0.0600,1.0000
C01376=90.850,12.420,106.000,0.0100,-0.0600,1.0000
C01377=81.060,11.260,102.250,0.0100,-0.0600,1.0000
C01378=73.410,10.270,98.450,0.0100,-0.0400,1.0000
C01379=68.760,8.660,95.630,-0.1700,0.1900,0.9700
C01380=67.430,4.900,94.500,-0.4600,0.0600,0.8900
C01381=67.460,1.980,94.450,-0.4800,-0.0200,0.8800
C01382=67.480,0.000,94.480,-0.4800,-0.0000,0.8800
C01383=67.460,-1.980,94.450,-0.4800,0.0200,0.8800
C01384=67.430,-4.900,94.500,-0.4600,-0.0600,0.8900
C01385=68.760,-8.660,95.630,-0.1700,-0.1900,0.9700
C01386=73.410,-10.270,98.450,0.0100,0.0400,1.0000
C01387=81.060,-11.260,102.250,0.0100,0.0600,1.0000
C01388=90.850,-12.420,106.000,0.0100,0.0600,1.0000
C01389=101.300,-13.690,108.730,0.0100,0.0600,1.0000
C01390=110.670,-15.110,110.040,0.0200,0.0500,1.0000
C01391=117.490,-19.610,110.710,0.0300,0.0200,1.0000
C01392=120.820,-26.730,111.250,0.0200,0.0000,1.0000
C01393=120.000,-34.990,111.800,0.0000,-0.0000,1.0000
C01394=117.170,-43.550,112.150,0.0000,-0.0000,1.0000
C01395=113.640,-52.060,112.150,0.0000,-0.0000,1.0000
C01396=109.590,-60.110,111.800,0.0000,-0.0000,1.0000
C01397=104.340,-66.530,111.250,0.0100,-0.0100,1.0000
C01398=96.950,-69.210,110.710,0.0000,-0.0300,1.0000
C01399=88.950,-67.570,110.040,-0.0300,-0.0500,1.0000
C01400=81.310,-61.950,108.730,-0.0400,-0.0500,1.0000
C01401=73.020,-55.460,106.000,-0.0400,-0.0500,1.0000
C01402=65.280,-49.360,102.250,-0.0300,-0.0500,1.0000
C01403=59.170,-44.640,98.450,-0.0200,-0.0300,1.0000
C01404=54.750,-42.500,95.630,0.0100,0.2500,0.9700
C01405=51.140,-44.220,94.500,-0.2800,0.3700,0.8900
C01406=49.110,-46.300,94.450,-0.3500,0.3200,0.8800
C01407=47.720,-47.720,94.480,-0.3400,0.3400,0.8800
C01408=46.300,-49.110,94.450,-0.3200,0.3500,0.8800
C01409=44.220,-51.140,94.500,-0.3700,0.2800,0.8900
C01410=42.500,-54.750,95.630,-0.2500,-0.0100,0.9700
C01411=44.640,-59.170,98.450,0.0300,0.0200,1.0000
C01412=49.360,-65.280,102.250,0.0500,0.0300,1.0000
C01413=55.460,-73.020,106.000,0.0500,0.0400,1.0000
C01414=61.950,-81.310,108.730,0.0500,0.0400,1.0000
C01415=67.570,-88.950,110.040,0.0500,0.0300,1.0000
C01416=69.210,-96.950,110.710,0.0300,-0.0000,1.0000
C01417=66.530,-104.340,111.250,0.0100,-0.0100,1.0000
C01418=60.110,-109.590,111.800,0.0000,-0.0000,1.0000
C01419=52.060,-113.640,112.150,0.0000,-0.0000,1.0000
C01420=43.550,-117.170,112.150,0.0000,-0.0000,1.0000
C01421=34.990,-120.000,111.800,0.0000,-0.0000,1.0000
C01422=26.730,-120.820,111.250,-0.0000,-0.0200,1.0000
C01423=19.610,-117.490,110.710,-0.0200,-0.0300,1.0000
C01424=15.110,-110.670,110.040,-0.0500,-0.0200,1.0000
C01425=13.690,-101.300,108.730,-0.0600,-0.0100,1.0000
C01426=12.420,-90.850,106.000,-0.0600,-0.0100,1.0000
C01427=11.260,-81.060,102.250,-0.0600,-0.0100,1.0000
C01428=10.270,-73.410,98.450,-0.0400,-0.0100,1.0000
C01429=8.660,-68.760,95.630,0.1900,0.1700,0.9700
C01430=4.900,-67.430,94.500,0.0600,0.4600,0.8900
C01431=1.980,-67.460,94.450,-0.0200,0.4800,0.8800
C01432=0.000,-67.480,94.480,-0.0000,0.4800,0.8800
C01433=0.000,-67.480,94.480,-0.0000,0.4800,0.8800
C01434=-1.980,-67.460,94.450,0.0200,0.4800,0.8800
C01435=-4.900,-67.430,94.500,-0.0600,0.4600,0.8900
C01436=-8.660,-68.760,95.630,-0.1900,0.1700,0.9700
C01437=-10.270,-73.410,98.450,0.0400,-0.0100,1.0000
C01438=-11.260,-81.060,102.250,0.0600,-0.0100,1.0000
C01439=-12.420,-90.850,106.000,0.0600,-0.0100,1.0000
C01440=-13.690,-101.300,108.730,0.0600,-0.0100,1.0000
C01441=-15.110,-110.670,110.040,0.0500,-0.0200,1.0000
C01442=-19.610,-117.490,110.710,0.0200,-0.0300,1.0000
C01443=-26.730,-120.820,111.250,0.0000,-0.0200,1.0000
C01444=-34.990,-120.000,111.800,-0.0000,-0.0000,1.0000
C01445=-43.550,-117.170,112.150,-0.0000,-0.0000,1.0000
C01446=-52.060,-113.640,112.150,-0.0000,-0.0000,1.0000
C01447=-60.110,-109.590,111.800,-0.0000,-0.0000,1.0000
C01448=-66.530,-104.340,111.250,-0.0100,-0.0100,1.0000
C01449=-69.210,-96.950,110.710,-0.0300,-0.0000,1.0000
C01450=-67.570,-88.950,110.040,-0.0500,0.0300,1.0000
C01451=-61.950,-81.310,108.730,-0.0500,0.0400,1.0000
C01452=-55.460,-73.020,106.000,-0.0500,0.0400,1.0000
C01453=-49.360,-65.280,102.250,-0.0500,0.0300,1.0000
C01454=-44.640,-59.170,98.450,-0.0300,0.0200,1.0000
C01455=-42.500,-54.750,95.630,0.2500,-0.0100,0.9700
C01456=-44.220,-51.140,94.500,0.3700,0.2800,0.8900
C01457=-46.300,-49.110,94.450,0.3200,0.3500,0.8800
C01458=-47.720,-47.720,94.480,0.3400,0.3400,0.8800
C01459=-49.110,-46.300,94.450,0.3500,0.3200,0.8800
C01460=-51.140,-44.220,94.500,0.2800,0.3700,0.8900
C01461=-54.750,-42.500,95.630,-0.0100,0.2500,0.9700
C01462=-59.170,-44.640,98.450,0.0200,-0.0300,1.0000
C01463=-65.280,-49.360,102.250,0.0300,-0.0500,1.0000
C01464=-73.020,-55.460,106.000,0.0400,-0.0500,1.0000
C01465=-81.310,-61.950,108.730,0.0400,-0.0500,1.0000
C01466=-88.950,-67.570,110.040,0.0300,-0.0500,1.0000
C01467=-96.950,-69.210,110.710,-0.0000,-0.0300,1.0000
C01468=-104.340,-66.530,111.250,-0.0100,-0.0100,1.0000
C01469=-109.590,-60.110,111.800,-0.0000,-0.0000,1.0000
C01470=-113.640,-52.060,112.150,-0.0000,-0.0000,1.0000
C01471=-117.170,-43.550,112.150,-0.0000,-0.0000,1.0000
C01472=-120.000,-34.990,111.800,-0.0000,-0.0000,1.0000
C01473=-120.820,-26.730,111.250,-0.0200,0.0000,1.0000
C01474=-117.490,-19.610,110.710,-0.0300,0.0200,1.0000
C01475=-110.670,-15.110,110.040,-0.0200,0.0500,1.0000
C01476=-101.300,-13.690,108.730,-0.0100,0.0600,1.0000
C01477=-90.850,-12.420,106.000,-0.0100,0.0600,1.0000
C01478=-81.060,-11.260,102.250,-0.0100,0.0600,1.0000
C01479=-73.410,-10.270,98.450,-0.0100,0.0400,1.0000
C01480=-68.760,-8.660,95.630,0.1700,-0.1900,0.9700
C01481=-67.430,-4.900,94.500,0.4600,-0.0600,0.8900
C01482=-67.460,-1.980,94.450,0.4800,0.0200,0.8800
C01483=-67.480,0.000,94.480,0.4800,0.0000,0.8800
C01484=-67.460,1.980,94.450,0.4800,-0.0200,0.8800
C01485=-67.430,4.900,94.500,0.4600,0.0600,0.8900
C01486=-68.760,8.660,95.630,0.1700,0.1900,0.9700
C01487=-73.410,10.270,98.450,-0.0100,-0.0400,1.0000
C01488=-81.060,11.260,102.250,-0.0100,-0.0600,1.0000
C01489=-90.850,12.420,106.000,-0.0100,-0.0600,1.0000
C01490=-101.300,13.690,108.730,-0.0100,-0.0600,1.0000
C01491=-110.670,15.110,110.040,-0.0200,-0.0500,1.0000
C01492=-117.490,19.610,110.710,-0.0300,-0.0200,1.0000
C01493=-120.820,26.730,111.250,-0.0200,-0.0000,1.0000
C01494=-120.000,34.990,111.800,-0.0000,0.0000,1.0000
C01495=-117.170,43.550,112.150,-0.0000,0.0000,1.0000
C01496=-113.640,52.060,112.150,-0.0000,0.0000,1.0000
C01497=-109.590,60.110,111.800,-0.0000,0.0000,1.0000
C01498=-104.340,66.530,111.250,-0.0100,0.0100,1.0000
C01499=-96.950,69.210,110.710,-0.0000,0.0300,1.0000
C01500=-88.950,67.570,110.040,0.0300,0.0500,1.0000
C01501=-81.310,61.950,108.730,0.0400,0.0500,1.0000
C01502=-73.020,55.460,106.000,0.0400,0.0500,1.0000
C01503=-65.280,49.360,102.250,0.0300,0.0500,1.0000
C01504=-59.170,44.640,98.450,0.0200,0.0300,1.0000
C01505=-54.750,42.500,95.630,-0.0100,-0.2500,0.9700
C01506=-51.140,44.220,94.500,0.2800,-0.3700,0.8900
C01507=-49.110,46.300,94.450,0.3500,-0.3200,0.8800
C01508=-47.720,47.720,94.480,0.3400,-0.3400,0.8800
C01509=-46.300,49.110,94.450,0.3200,-0.3500,0.8800
C01510=-44.220,51.140,94.500,0.3700,-0.2800,0.8900
C01511=-42.500,54.750,95.630,0.2500,0.0100,0.9700
C01512=-44.640,59.170,98.450,-0.0300,-0.0200,1.0000
C01513=-49.360,65.280,102.250,-0.0500,-0.0300,1.0000
C01514=-55.460,73.020,106.000,-0.0500,-0.0400,1.0000
C01515=-61.950,81.310,108.730,-0.0500,-0.0400,1.0000
C01516=-67.570,88.950,110.040,-0.0500,-0.0300,1.0000
C01517=-69.210,96.950,110.710,-0.0300,0.0000,1.0000
C01518=-66.530,104.340,111.250,-0.0100,0.0100,1.0000
C01519=-60.110,109.590,111.800,-0.0000,0.0000,1.0000
C01520=-52.060,113.640,112.150,-0.0000,0.0000,1.0000
C01521=-43.550,117.170,112.150,-0.0000,0.0000,1.0000
C01522=-34.990,120.000,111.800,-0.0000,0.0000,1.0000
C01523=-26.730,120.820,111.250,0.0000,0.0200,1.0000
C01524=-19.610,117.490,110.710,0.0200,0.0300,1.0000
C01525=-15.110,110.670,110.040,0.0500,0.0200,1.0000
C01526=-13.690,101.300,108.730,0.0600,0.0100,1.0000
C01527=-12.420,90.850,106.000,0.0600,0.0100,1.0000
C01528=-11.260,81.060,102.250,0.0600,0.0100,1.0000
C01529=-10.270,73.410,98.450,0.0400,0.0100,1.0000
C01530=-8.660,68.760,95.630,-0.1900,-0.1700,0.9700
C01531=-4.900,67.430,94.500,-0.0600,-0.4600,0.8900
C01532=-1.980,67.460,94.450,0.0200,-0.4800,0.8800
C01533=0.000,67.480,94.480,-0.0000,-0.4800,0.8800
C01534=0.000,66.690,95.980,-0.0000,-0.4600,0.8900
C01535=-1.910,66.670,95.950,0.0200,-0.4600,0.8900
C01536=-4.770,66.650,96.000,-0.0600,-0.4400,0.9000
C01537=-8.520,68.030,97.160,-0.1800,-0.1600,0.9700
C01538=-10.110,72.800,100.040,0.0400,0.0100,1.0000
C01539=-11.100,80.630,103.890,0.0500,0.0100,1.0000
C01540=-12.280,90.580,107.670,0.0500,0.0100,1.0000
C01541=-13.580,101.170,110.420,0.0500,0.0100,1.0000
C01542=-15.000,110.620,111.730,0.0400,0.0100,1.0000
C01543=-19.520,117.480,112.410,0.0200,0.0200,1.0000
C01544=-26.660,120.840,112.950,0.0000,0.0100,1.0000
C01545=-34.950,120.010,113.500,-0.0000,0.0000,1.0000
C01546=-43.530,117.170,113.850,-0.0000,0.0000,1.0000
C01547=-52.070,113.640,113.850,-0.0000,0.0000,1.0000
C01548=-60.150,109.580,113.500,-0.0000,0.0000,1.0000
C01549=-66.590,104.300,112.950,-0.0100,0.0100,1.0000
C01550=-69.270,96.870,112.410,-0.0300,0.0000,1.0000
C01551=-67.610,88.830,111.730,-0.0400,-0.0200,1.0000
C01552=-61.930,81.140,110.420,-0.0400,-0.0300,1.0000
C01553=-55.370,72.740,107.670,-0.0400,-0.0300,1.0000
C01554=-49.170,64.870,103.890,-0.0400,-0.0300,1.0000
C01555=-44.330,58.630,100.040,-0.0300,-0.0200,1.0000
C01556=-42.080,54.130,97.160,0.2400,0.0100,0.9700
C01557=-43.750,50.500,96.000,0.3500,-0.2700,0.9000
C01558=-45.790,48.490,95.950,0.3100,-0.3400,0.8900
C01559=-47.150,47.150,95.980,0.3200,-0.3200,0.8900
C01560=-48.490,45.790,95.950,0.3400,-0.3100,0.8900
C01561=-50.500,43.750,96.000,0.2700,-0.3500,0.9000
C01562=-54.130,42.080,97.160,-0.0100,-0.2400,0.9700
C01563=-58.630,44.330,100.040,0.0200,0.0300,1.0000
C01564=-64.870,49.170,103.890,0.0300,0.0400,1.0000
C01565=-72.740,55.370,107.670,0.0300,0.0400,1.0000
C01566=-81.140,61.930,110.420,0.0300,0.0400,1.0000
C01567=-88.830,67.610,111.730,0.0200,0.0400,1.0000
C01568=-96.870,69.270,112.410,-0.0000,0.0300,1.0000
C01569=-104.300,66.590,112.950,-0.0100,0.0100,1.0000
C01570=-109.580,60.150,113.500,-0.0000,0.0000,1.0000
C01571=-113.640,52.070,113.850,-0.0000,0.0000,1.0000
C01572=-117.170,43.530,113.850,-0.0000,0.0000,1.0000
C01573=-120.010,34.950,113.500,-0.0000,0.0000,1.0000
C01574=-120.840,26.660,112.950,-0.0100,-0.0000,1.0000
C01575=-117.480,19.520,112.410,-0.0200,-0.0200,1.0000
C01576=-110.620,15.000,111.730,-0.0100,-0.0400,1.0000
C01577=-101.170,13.580,110.420,-0.0100,-0.0500,1.0000
C01578=-90.580,12.280,107.670,-0.0100,-0.0500,1.0000
C01579=-80.630,11.100,103.890,-0.0100,-0.0500,1.0000
C01580=-72.800,10.110,100.040,-0.0100,-0.0400,1.0000
C01581=-68.030,8.520,97.160,0.1600,0.1800,0.9700
C01582=-66.650,4.770,96.000,0.4400,0.0600,0.9000
C01583=-66.670,1.910,95.950,0.4600,-0.0200,0.8900
C01584=-66.690,0.000,95.980,0.4600,0.0000,0.8900
C01585=-66.670,-1.910,95.950,0.4600,0.0200,0.8900
C01586=-66.650,-4.770,96.000,0.4400,-0.0600,0.9000
C01587=-68.030,-8.520,97.160,0.1600,-0.1800,0.9700
C01588=-72.800,-10.110,100.040,-0.0100,0.0400,1.0000
C01589=-80.630,-11.100,103.890,-0.0100,0.0500,1.0000
C01590=-90.580,-12.280,107.670,-0.0100,0.0500,1.0000
C01591=-101.170,-13.580,110.420,-0.0100,0.0500,1.0000
C01592=-110.620,-15.000,111.730,-0.0100,0.0400,1.0000
C01593=-117.480,-19.520,112.410,-0.0200,0.0200,1.0000
C01594=-120.840,-26.660,112.950,-0.0100,0.0000,1.0000
C01595=-120.010,-34.950,113.500,-0.0000,-0.0000,1.0000
C01596=-117.170,-43.530,113.850,-0.0000,-0.0000,1.0000
C01597=-113.640,-52.070,113.850,-0.0000,-0.0000,1.0000
C01598=-109.580,-60.150,113.500,-0.0000,-0.0000,1.0000
C01599=-104.300,-66.590,112.950,-0.0100,-0.0100,1.0000
C01600=-96.870,-69.270,112.410,-0.0000,-0.0300,1.0000
C01601=-88.830,-67.610,111.730,0.0200,-0.0400,1.0000
C01602=-81.140,-61.930,110.420,0.0300,-0.0400,1.0000
C01603=-72.740,-55.370,107.670,0.0300,-0.0400,1.0000
C01604=-64.870,-49.170,103.890,0.0300,-0.0400,1.0000
C01605=-58.630,-44.330,100.040,0.0200,-0.0300,1.0000
C01606=-54.130,-42.080,97.160,-0.0100,0.2400,0.9700
C01607=-50.500,-43.750,96.000,0.2700,0.3500,0.9000
C01608=-48.490,-45.790,95.950,0.3400,0.3100,0.8900
C01609=-47.150,-47.150,95.980,0.3200,0.3200,0.8900
C01610=-45.790,-48.490,95.950,0.3100,0.3400,0.8900
C01611=-43.750,-50.500,96.000,0.3500,0.2700,0.9000
C01612=-42.080,-54.130,97.160,0.2400,-0.0100,0.9700
C01613=-44.330,-58.630,100.040,-0.0300,0.0200,1.0000
C01614=-49.170,-64.870,103.890,-0.0400,0.0300,1.0000
C01615=-55.370,-72.740,107.670,-0.0400,0.0300,1.0000
C01616=-61.930,-81.140,110.420,-0.0400,0.0300,1.0000
C01617=-67.610,-88.830,111.730,-0.0400,0.0200,1.0000
C01618=-69.270,-96.870,112.410,-0.0300,-0.0000,1.0000
C01619=-66.590,-104.300,112.950,-0.0100,-0.0100,1.0000
C01620=-60.150,-109.580,113.500,-0.0000,-0.0000,1.0000
C01621=-52.070,-113.640,113.850,-0.0000,-0.0000,1.0000
C01622=-43.530,-117.170,113.850,-0.0000,-0.0000,1.0000
C01623=-34.950,-120.010,113.500,-0.0000,-0.0000,1.0000
C01624=-26.660,-120.840,112.950,0.0000,-0.0100,1.0000
C01625=-19.520,-117.480,112.410,0.0200,-0.0200,1.0000
C01626=-15.000,-110.620,111.730,0.0400,-0.0100,1.0000
C01627=-13.580,-101.170,110.420,0.0500,-0.0100,1.0000
C01628=-12.280,-90.580,107.670,0.0500,-0.0100,1.0000
C01629=-11.100,-80.630,103.890,0.0500,-0.0100,1.0000
C01630=-10.110,-72.800,100.040,0.0400,-0.0100,1.0000
C01631=-8.520,-68.030,97.160,-0.1800,0.1600,0.9700
C01632=-4.770,-66.650,96.000,-0.0600,0.4400,0.9000
C01633=-1.910,-66.670,95.950,0.0200,0.4600,0.8900
C01634=0.000,-66.690,95.980,-0.0000,0.4600,0.8900
C01635=0.000,-66.690,95.980,-0.0000,0.4600,0.8900
C01636=1.910,-66.670,95.950,-0.0200,0.4600,0.8900
C01637=4.770,-66.650,96.000,0.0600,0.4400,0.9000
C01638=8.520,-68.030,97.160,0.1800,0.1600,0.9700
C01639=10.110,-72.800,100.040,-0.0400,-0.0100,1.0000
C01640=11.100,-80.630,103.890,-0.0500,-0.0100,1.0000
C01641=12.280,-90.580,107.670,-0.0500,-0.0100,1.0000
C01642=13.580,-101.170,110.420,-0.0500,-0.0100,1.0000
C01643=15.000,-110.620,111.730,-0.0400,-0.0100,1.0000
C01644=19.520,-117.480,112.410,-0.0200,-0.0200,1.0000
C01645=26.660,-120.840,112.950,-0.0000,-0.0100,1.0000
C01646=34.950,-120.010,113.500,0.0000,-0.0000,1.0000
C01647=43.530,-117.170,113.850,0.0000,-0.0000,1.0000
C01648=52.070,-113.640,113.850,0.0000,-0.0000,1.0000
C01649=60.150,-109.580,113.500,0.0000,-0.0000,1.0000
C01650=66.590,-104.300,112.950,0.0100,-0.0100,1.0000
C01651=69.270,-96.870,112.410,0.0300,-0.0000,1.0000
C01652=67.610,-88.830,111.730,0.0400,0.0200,1.0000
C01653=61.930,-81.140,110.420,0.0400,0.0300,1.0000
C01654=55.370,-72.740,107.670,0.0400,0.0300,1.0000
C01655=49.170,-64.870,103.890,0.0400,0.0300,1.0000
C01656=44.330,-58.630,100.040,0.0300,0.0200,1.0000
C01657=42.080,-54.130,97.160,-0.2400,-0.0100,0.9700
C01658=43.750,-50.500,96.000,-0.3500,0.2700,0.9000
C01659=45.790,-48.490,95.950,-0.3100,0.3400,0.8900
C01660=47.150,-47.150,95.980,-0.3200,0.3200,0.8900
C01661=48.490,-45.790,95.950,-0.3400,0.3100,0.8900
C01662=50.500,-43.750,96.000,-0.2700,0.3500,0.9000
C01663=54.130,-42.080,97.160,0.0100,0.2400,0.9700
C01664=58.630,-44.330,100.040,-0.0200,-0.0300,1.0000
C01665=64.870,-49.170,103.890,-0.0300,-0.0400,1.0000
C01666=72.740,-55.370,107.670,-0.0300,-0.0400,1.0000
C01667=81.140,-61.930,110.420,-0.0300,-0.0400,1.0000
C01668=88.830,-67.610,111.730,-0.0200,-0.0400,1.0000
C01669=96.870,-69.270,112.410,0.0000,-0.0300,1.0000
C01670=104.300,-66.590,112.950,0.0100,-0.0100,1.0000
C01671=109.580,-60.150,113.500,0.0000,-0.0000,1.0000
C01672=113.640,-52.070,113.850,0.0000,-0.0000,1.0000
C01673=117.170,-43.530,113.850,0.0000,-0.0000,1.0000
C01674=120.010,-34.950,113.500,0.0000,-0.0000,1.0000
C01675=120.840,-26.660,112.950,0.0100,0.0000,1.0000
C01676=117.480,-19.520,112.410,0.0200,0.0200,1.0000
C01677=110.620,-15.000,111.730,0.0100,0.0400,1.0000
C01678=101.170,-13.580,110.420,0.0100,0.0500,1.0000
C01679=90.580,-12.280,107.670,0.0100,0.0500,1.0000
C01680=80.630,-11.100,103.890,0.0100,0.0500,1.0000
C01681=72.800,-10.110,100.040,0.0100,0.0400,1.0000
C01682=68.030,-8.520,97.160,-0.1600,-0.1800,0.9700
C01683=66.650,-4.770,96.000,-0.4400,-0.0600,0.9000
C01684=66.670,-1.910,95.950,-0.4600,0.0200,0.8900
C01685=66.690,0.000,95.980,-0.4600,-0.0000,0.8900
C01686=66.670,1.910,95.950,-0.4600,-0.0200,0.8900
C01687=66.650,4.770,96.000,-0.4400,0.0600,0.9000
C01688=68.030,8.520,97.160,-0.1600,0.1800,0.9700
C01689=72.800,10.110,100.040,0.0100,-0.0400,1.0000
C01690=80.630,11.100,103.890,0.0100,-0.0500,1.0000
C01691=90.580,12.280,107.670,0.0100,-0.0500,1.0000
C01692=101.170,13.580,110.420,0.0100,-0.0500,1.0000
C01693=110.620,15.000,111.730,0.0100,-0.0400,1.0000
C01694=117.480,19.520,112.410,0.0200,-0.0200,1.0000
C01695=120.840,26.660,112.950,0.0100,-0.0000,1.0000
C01696=120.010,34.950,113.500,0.0000,0.0000,1.0000
C01697=117.170,43.530,113.850,0.0000,0.0000,1.0000
C01698=113.640,52.070,113.850,0.0000,0.0000,1.0000
C01699=109.580,60.150,113.500,0.0000,0.0000,1.0000
C01700=104.300,66.590,112.950,0.0100,0.0100,1.0000
C01701=96.870,69.270,112.410,0.0000,0.0300,1.0000
C01702=88.830,67.610,111.730,-0.0200,0.0400,1.0000
C01703=81.140,61.930,110.420,-0.0300,0.0400,1.0000
C01704=72.740,55.370,107.670,-0.0300,0.0400,1.0000
C01705=64.870,49.170,103.890,-0.0300,0.0400,1.0000
C01706=58.630,44.330,100.040,-0.0200,0.0300,1.0000
C01707=54.130,42.080,97.160,0.0100,-0.2400,0.9700
C01708=50.500,43.750,96.000,-0.2700,-0.3500,0.9000
C01709=48.490,45.790,95.950,-0.3400,-0.3100,0.8900
C01710=47.150,47.150,95.980,-0.3200,-0.3200,0.8900
C01711=45.790,48.490,95.950,-0.3100,-0.3400,0.8900
C01712=43.750,50.500,96.000,-0.3500,-0.2700,0.9000
C01713=42.080,54.130,97.160,-0.2400,0.0100,0.9700
C01714=44.330,58.630,100.040,0.0300,-0.0200,1.0000
C01715=49.170,64.870,103.890,0.0400,-0.0300,1.0000
C01716=55.370,72.740,107.670,0.0400,-0.0300,1.0000
C01717=61.930,81.140,110.420,0.0400,-0.0300,1.0000
C01718=67.610,88.830,111.730,0.0400,-0.0200,1.0000
C01719=69.270,96.870,112.410,0.0300,0.0000,1.0000
C01720=66.590,104.300,112.950,0.0100,0.0100,1.0000
C01721=60.150,109.580,113.500,0.0000,0.0000,1.0000
C01722=52.070,113.640,113.850,0.0000,0.0000,1.0000
C01723=43.530,117.170,113.850,0.0000,0.0000,1.0000
C01724=34.950,120.010,113.500,0.0000,0.0000,1.0000
C01725=26.660,120.840,112.950,-0.0000,0.0100,1.0000
C01726=19.520,117.480,112.410,-0.0200,0.0200,1.0000
C01727=15.000,110.620,111.730,-0.0400,0.0100,1.0000
C01728=13.580,101.170,110.420,-0.0500,0.0100,1.0000
C01729=12.280,90.580,107.670,-0.0500,0.0100,1.0000
C01730=11.100,80.630,103.890,-0.0500,0.0100,1.0000
C01731=10.110,72.800,100.040,-0.0400,0.0100,1.0000
C01732=8.520,68.030,97.160,0.1800,-0.1600,0.9700
C01733=4.770,66.650,96.000,0.0600,-0.4400,0.9000
C01734=1.910,66.670,95.950,-0.0200,-0.4600,0.8900
C01735=0.000,66.690,95.980,-0.0000,-0.4600,0.8900
C01736=0.000,65.920,97.500,-0.0000,-0.4400,0.9000
C01737=1.840,65.910,97.470,-0.0100,-0.4400,0.9000
C01738=4.660,65.890,97.520,0.0600,-0.4200,0.9100
C01739=8.380,67.330,98.700,0.1700,-0.1500,0.9700
C01740=9.960,72.230,101.630,-0.0400,0.0100,1.0000
C01741=10.960,80.240,105.540,-0.0500,0.0100,1.0000
C01742=12.160,90.350,109.350,-0.0500,0.0100,1.0000
C01743=13.480,101.050,112.120,-0.0400,0.0100,1.0000
C01744=14.910,110.570,113.430,-0.0400,0.0100,1.0000
C01745=19.440,117.470,114.110,-0.0100,0.0200,1.0000
C01746=26.600,120.850,114.650,-0.0000,0.0100,1.0000
C01747=34.920,120.020,115.200,0.0000,0.0000,1.0000
C01748=43.520,117.180,115.550,0.0000,0.0000,1.0000
C01749=52.080,113.630,115.550,0.0000,0.0000,1.0000
C01750=60.180,109.560,115.200,0.0000,0.0000,1.0000
C01751=66.640,104.260,114.650,0.0100,0.0100,1.0000
C01752=69.320,96.810,114.110,0.0200,0.0000,1.0000
C01753=67.640,88.730,113.430,0.0300,-0.0200,1.0000
C01754=61.920,80.990,112.120,0.0300,-0.0300,1.0000
C01755=55.290,72.490,109.350,0.0400,-0.0300,1.0000
C01756=48.990,64.480,105.540,0.0400,-0.0300,1.0000
C01757=44.030,58.110,101.630,0.0300,-0.0200,1.0000
C01758=41.680,53.530,98.700,-0.2200,0.0100,0.9700
C01759=43.300,49.880,97.520,-0.3400,-0.2600,0.9100
C01760=45.300,47.900,97.470,-0.3000,-0.3200,0.9000
C01761=46.610,46.610,97.500,-0.3100,-0.3100,0.9000
C01762=47.900,45.300,97.470,-0.3200,-0.3000,0.9000
C01763=49.880,43.300,97.520,-0.2600,-0.3400,0.9100
C01764=53.530,41.680,98.700,0.0100,-0.2200,0.9700
C01765=58.110,44.030,101.630,-0.0200,0.0300,1.0000
C01766=64.480,48.990,105.540,-0.0300,0.0400,1.0000
C01767=72.490,55.290,109.350,-0.0300,0.0400,1.0000
C01768=80.990,61.920,112.120,-0.0300,0.0300,1.0000
C01769=88.730,67.640,113.430,-0.0200,0.0300,1.0000
C01770=96.810,69.320,114.110,0.0000,0.0200,1.0000
C01771=104.260,66.640,114.650,0.0100,0.0100,1.0000
C01772=109.560,60.180,115.200,0.0000,0.0000,1.0000
C01773=113.630,52.080,115.550,0.0000,0.0000,1.0000
C01774=117.180,43.520,115.550,0.0000,0.0000,1.0000
C01775=120.020,34.920,115.200,0.0000,0.0000,1.0000
C01776=120.850,26.600,114.650,0.0100,-0.0000,1.0000
C01777=117.470,19.440,114.110,0.0200,-0.0100,1.0000
C01778=110.570,14.910,113.430,0.0100,-0.0400,1.0000
C01779=101.050,13.480,112.120,0.0100,-0.0400,1.0000
C01780=90.350,12.160,109.350,0.0100,-0.0500,1.0000
C01781=80.240,10.960,105.540,0.0100,-0.0500,1.0000
C01782=72.230,9.960,101.630,0.0100,-0.0400,1.0000
C01783=67.330,8.380,98.700,-0.1500,0.1700,0.9700
C01784=65.890,4.660,97.520,-0.4200,0.0600,0.9100
C01785=65.910,1.840,97.470,-0.4400,-0.0100,0.9000
C01786=65.920,0.000,97.500,-0.4400,-0.0000,0.9000
C01787=65.910,-1.840,97.470,-0.4400,0.0100,0.9000
C01788=65.890,-4.660,97.520,-0.4200,-0.0600,0.9100
C01789=67.330,-8.380,98.700,-0.1500,-0.1700,0.9700
C01790=72.230,-9.960,101.630,0.0100,0.0400,1.0000
C01791=80.240,-10.960,105.540,0.0100,0.0500,1.0000
C01792=90.350,-12.160,109.350,0.0100,0.0500,1.0000
C01793=101.050,-13.480,112.120,0.0100,0.0400,1.0000
C01794=110.570,-14.910,113.430,0.0100,0.0400,1.0000
C01795=117.470,-19.440,114.110,0.0200,0.0100,1.0000
C01796=120.850,-26.600,114.650,0.0100,0.0000,1.0000
C01797=120.020,-34.920,115.200,0.0000,-0.0000,1.0000
C01798=117.180,-43.520,115.550,0.0000,-0.0000,1.0000
C01799=113.630,-52.080,115.550,0.0000,-0.0000,1.0000
C01800=109.560,-60.180,115.200,0.0000,-0.0000,1.0000
C01801=104.260,-66.640,114.650,0.0100,-0.0100,1.0000
C01802=96.810,-69.320,114.110,0.0000,-0.0200,1.0000
C01803=88.730,-67.640,113.430,-0.0200,-0.0300,1.0000
C01804=80.990,-61.920,112.120,-0.0300,-0.0300,1.0000
C01805=72.490,-55.290,109.350,-0.0300,-0.0400,1.0000
C01806=64.480,-48.990,105.540,-0.0300,-0.0400,1.0000
C01807=58.110,-44.030,101.630,-0.0200,-0.0300,1.0000
C01808=53.530,-41.680,98.700,0.0100,0.2200,0.9700
C01809=49.880,-43.300,97.520,-0.2600,0.3400,0.9100
C01810=47.900,-45.300,97.470,-0.3200,0.3000,0.9000
C01811=46.610,-46.610,97.500,-0.3100,0.3100,0.9000
C01812=45.300,-47.900,97.470,-0.3000,0.3200,0.9000
C01813=43.300,-49.880,97.520,-0.3400,0.2600,0.9100
C01814=41.680,-53.530,98.700,-0.2200,-0.0100,0.9700
C01815=44.030,-58.110,101.630,0.0300,0.0200,1.0000
C01816=48.990,-64.480,105.540,0.0400,0.0300,1.0000
C01817=55.290,-72.490,109.350,0.0400,0.0300,1.0000
C01818=61.920,-80.990,112.120,0.0300,0.0300,1.0000
C01819=67.640,-88.730,113.430,0.0300,0.0200,1.0000
C01820=69.320,-96.810,114.110,0.0200,-0.0000,1.0000
C01821=66.640,-104.260,114.650,0.0100,-0.0100,1.0000
C01822=60.180,-109.560,115.200,0.0000,-0.0000,1.0000
C01823=52.080,-113.630,115.550,0.0000,-0.0000,1.0000
C01824=43.520,-117.180,115.550,0.0000,-0.0000,1.0000
C01825=34.920,-120.020,115.200,0.0000,-0.0000,1.0000
C01826=26.600,-120.850,114.650,-0.0000,-0.0100,1.0000
C01827=19.440,-117.470,114.110,-0.0100,-0.0200,1.0000
C01828=14.910,-110.570,113.430,-0.0400,-0.0100,1.0000
C01829=13.480,-101.050,112.120,-0.0400,-0.0100,1.0000
C01830=12.160,-90.350,109.350,-0.0500,-0.0100,1.0000
C01831=10.960,-80.240,105.540,-0.0500,-0.0100,1.0000
C01832=9.960,-72.230,101.630,-0.0400,-0.0100,1.0000
C01833=8.380,-67.330,98.700,0.1700,0.1500,0.9700
C01834=4.660,-65.890,97.520,0.0600,0.4200,0.9100
C01835=1.840,-65.910,97.470,-0.0100,0.4400,0.9000
C01836=0.000,-65.920,97.500,-0.0000,0.4400,0.9000
C01837=0.000,-65.920,97.500,-0.0000,0.4400,0.9000
C01838=-1.840,-65.910,97.470,0.0100,0.4400,0.9000
C01839=-4.660,-65.890,97.520,-0.0600,0.4200,0.9100
C01840=-8.380,-67.330,98.700,-0.1700,0.1500,0.9700
C01841=-9.960,-72.230,101.630,0.0400,-0.0100,1.0000
C01842=-10.960,-80.240,105.540,0.0500,-0.0100,1.0000
C01843=-12.160,-90.350,109.350,0.0500,-0.0100,1.0000
C01844=-13.480,-101.050,112.120,0.0400,-0.0100,1.0000
C01845=-14.910,-110.570,113.430,0.0400,-0.0100,1.0000
C01846=-19.440,-117.470,114.110,0.0100,-0.0200,1.0000
C01847=-26.600,-120.850,114.650,0.0000,-0.0100,1.0000
C01848=-34.920,-120.020,115.200,-0.0000,-0.0000,1.0000
C01849=-43.520,-117.180,115.550,-0.0000,-0.0000,1.0000
C01850=-52.080,-113.630,115.550,-0.0000,-0.0000,1.0000
C01851=-60.180,-109.560,115.200,-0.0000,-0.0000,1.0000
C01852=-66.640,-104.260,114.650,-0.0100,-0.0100,1.0000
C01853=-69.320,-96.810,114.110,-0.0200,-0.0000,1.0000
C01854=-67.640,-88.730,113.430,-0.0300,0.0200,1.0000
C01855=-61.920,-80.990,112.120,-0.0300,0.0300,1.0000
C01856=-55.290,-72.490,109.350,-0.0400,0.0300,1.0000
C01857=-48.990,-64.480,105.540,-0.0400,0.0300,1.0000
C01858=-44.030,-58.110,101.630,-0.0300,0.0200,1.0000
C01859=-41.680,-53.530,98.700,0.2200,-0.0100,0.9700
C01860=-43.300,-49.880,97.520,0.3400,0.2600,0.9100
C01861=-45.300,-47.900,97.470,0.3000,0.3200,0.9000
C01862=-46.610,-46.610,97.500,0.3100,0.3100,0.9000
C01863=-47.900,-45.300,97.470,0.3200,0.3000,0.9000
C01864=-49.880,-43.300,97.520,0.2600,0.3400,0.9100
C01865=-53.530,-41.680,98.700,-0.0100,0.2200,0.9700
C01866=-58.110,-44.030,101.630,0.0200,-0.0300,1.0000
C01867=-64.480,-48.990,105.540,0.0300,-0.0400,1.0000
C01868=-72.490,-55.290,109.350,0.0300,-0.0400,1.0000
C01869=-80.990,-61.920,112.120,0.0300,-0.0300,1.0000
C01870=-88.730,-67.640,113.430,0.0200,-0.0300,1.0000
C01871=-96.810,-69.320,114.110,-0.0000,-0.0200,1.0000
C01872=-104.260,-66.640,114.650,-0.0100,-0.0100,1.0000
C01873=-109.560,-60.180,115.200,-0.0000,-0.0000,1.0000
C01874=-113.630,-52.080,115.550,-0.0000,-0.0000,1.0000
C01875=-117.180,-43.520,115.550,-0.0000,-0.0000,1.0000
C01876=-120.020,-34.920,115.200,-0.0000,-0.0000,1.0000
C01877=-120.850,-26.600,114.650,-0.0100,0.0000,1.0000
C01878=-117.470,-19.440,114.110,-0.0200,0.0100,1.0000
C01879=-110.570,-14.910,113.430,-0.0100,0.0400,1.0000
C01880=-101.050,-13.480,112.120,-0.0100,0.0400,1.0000
C01881=-90.350,-12.160,109.350,-0.0100,0.0500,1.0000
C01882=-80.240,-10.960,105.540,-0.0100,0.0500,1.0000
C01883=-72.230,-9.960,101.630,-0.0100,0.0400,1.0000
C01884=-67.330,-8.380,98.700,0.1500,-0.1700,0.9700
C01885=-65.890,-4.660,97.520,0.4200,-0.0600,0.9100
C01886=-65.910,-1.840,97.470,0.4400,0.0100,0.9000
C01887=-65.920,0.000,97.500,0.4400,0.0000,0.9000
C01888=-65.910,1.840,97.470,0.4400,-0.0100,0.9000
C01889=-65.890,4.660,97.520,0.4200,0.0600,0.9100
C01890=-67.330,8.380,98.700,0.1500,0.1700,0.9700
C01891=-72.230,9.960,101.630,-0.0100,-0.0400,1.0000
C01892=-80.240,10.960,105.540,-0.0100,-0.0500,1.0000
C01893=-90.350,12.160,109.350,-0.0100,-0.0500,1.0000
C01894=-101.050,13.480,112.120,-0.0100,-0.0400,1.0000
C01895=-110.570,14.910,113.430,-0.0100,-0.0400,1.0000
C01896=-117.470,19.440,114.110,-0.0200,-0.0100,1.0000
C01897=-120.850,26.600,114.650,-0.0100,-0.0000,1.0000
C01898=-120.020,34.920,115.200,-0.0000,0.0000,1.0000
C01899=-117.180,43.520,115.550,-0.0000,0.0000,1.0000
C01900=-113.630,52.080,115.550,-0.0000,0.0000,1.0000
C01901=-109.560,60.180,115.200,-0.0000,0.0000,1.0000
C01902=-104.260,66.640,114.650,-0.0100,0.0100,1.0000
C01903=-96.810,69.320,114.110,-0.0000,0.0200,1.0000
C01904=-88.730,67.640,113.430,0.0200,0.0300,1.0000
C01905=-80.990,61.920,112.120,0.0300,0.0300,1.0000
C01906=-72.490,55.290,109.350,0.0300,0.0400,1.0000
C01907=-64.480,48.990,105.540,0.0300,0.0400,1.0000
C01908=-58.110,44.030,101.630,0.0200,0.0300,1.0000
C01909=-53.530,41.680,98.700,-0.0100,-0.2200,0.9700
C01910=-49.880,43.300,97.520,0.2600,-0.3400,0.9100
C01911=-47.900,45.300,97.470,0.3200,-0.3000,0.9000
C01912=-46.610,46.610,97.500,0.3100,-0.3100,0.9000
C01913=-45.300,47.900,97.470,0.3000,-0.3200,0.9000
C01914=-43.300,49.880,97.520,0.3400,-0.2600,0.9100
C01915=-41.680,53.530,98.700,0.2200,0.0100,0.9700
C01916=-44.030,58.110,101.630,-0.0300,-0.0200,1.0000
C01917=-48.990,64.480,105.540,-0.0400,-0.0300,1.0000
C01918=-55.290,72.490,109.350,-0.0400,-0.0300,1.0000
C01919=-61.920,80.990,112.120,-0.0300,-0.0300,1.0000
C01920=-67.640,88.730,113.430,-0.0300,-0.0200,1.0000
C01921=-69.320,96.810,114.110,-0.0200,0.0000,1.0000
C01922=-66.640,104.260,114.650,-0.0100,0.0100,1.0000
C01923=-60.180,109.560,115.200,-0.0000,0.0000,1.0000
C01924=-52.080,113.630,115.550,-0.0000,0.0000,1.0000
C01925=-43.520,117.180,115.550,-0.0000,0.0000,1.0000
